LIN {X 0,Y 405.524,Z 705.596,A -85,B 0,C 180,E1 17049.688,E2 17049.688} C_VEL
LIN {X 0,Y 402.242,Z 726.337,A -85,B 0,C 180,E1 17048.422,E2 17048.422} C_VEL
LIN {X 0,Y 398.508,Z 746.053,A -85,B 0,C 180,E1 17046.936,E2 17046.936} C_VEL
LIN {X 0,Y 394.229,Z 765.506,A -85,B 0,C 180,E1 17045.152,E2 17045.152} C_VEL
LIN {X 0,Y 389.705,Z 783.802,A -85,B 0,C 180,E1 17043.128,E2 17043.128} C_VEL
LIN {X 0,Y 385.137,Z 800.764,A -85,B 0,C 180,E1 17040.878,E2 17040.878} C_VEL
LIN {X 0,Y 380.552,Z 816.747,A -85,B 0,C 180,E1 17038.332,E2 17038.332} C_VEL
LIN {X 0,Y 376.385,Z 830.752,A -85,B 0,C 180,E1 17035.659,E2 17035.659} C_VEL
LIN {X 0,Y 372.544,Z 843.468,A -85,B 0,C 180,E1 17032.736,E2 17032.736} C_VEL
LIN {X 0,Y 369.226,Z 854.588,A -85,B 0,C 180,E1 17029.621,E2 17029.621} C_VEL
LIN {X 0,Y 366.629,Z 863.669,A -85,B 0,C 180,E1 17026.477,E2 17026.477} C_VEL
LIN {X 0,Y 364.673,Z 871.061,A -85,B 0,C 180,E1 17023.251,E2 17023.251} C_VEL
LIN {X 0,Y 363.308,Z 876.769,A -85,B 0,C 180,E1 17019.985,E2 17019.985} C_VEL
LIN {X 0,Y 362.432,Z 881.033,A -85,B 0,C 180,E1 17016.495,E2 17016.495} C_VEL
LIN {X 0,Y 362.034,Z 883.325,A -85,B 0,C 180,E1 17013.417,E2 17013.417} C_VEL
LIN {X 0,Y 360.957,Z 883.954,A -85,B 0,C 180,E1 17012.201,E2 17012.201} C_VEL
LIN {X 0,Y 354.617,Z 885.109,A -85,B 0,C 180,E1 17008.857,E2 17008.857} C_VEL
LIN {X 0,Y 354.012,Z 884.908,A -85,B 0,C 180,E1 17007.87,E2 17007.87} C_VEL
LIN {X 0,Y 354.34,Z 883.134,A -85,B 0,C 180,E1 17004.495,E2 17004.495} C_VEL
LIN {X 0,Y 355.032,Z 879.694,A -85,B 0,C 180,E1 17001.089,E2 17001.089} C_VEL
LIN {X 0,Y 356.194,Z 874.854,A -85,B 0,C 180,E1 16997.846,E2 16997.846} C_VEL
LIN {X 0,Y 358.029,Z 868.036,A -85,B 0,C 180,E1 16994.449,E2 16994.449} C_VEL
LIN {X 0,Y 360.466,Z 859.76,A -85,B 0,C 180,E1 16991.23,E2 16991.23} C_VEL
LIN {X 0,Y 363.449,Z 850.138,A -85,B 0,C 180,E1 16988.198,E2 16988.198} C_VEL
LIN {X 0,Y 367.117,Z 838.547,A -85,B 0,C 180,E1 16985.201,E2 16985.201} C_VEL
LIN {X 0,Y 371.487,Z 824.659,A -85,B 0,C 180,E1 16982.248,E2 16982.248} C_VEL
LIN {X 0,Y 376.128,Z 809.477,A -85,B 0,C 180,E1 16979.574,E2 16979.574} C_VEL
LIN {X 0,Y 380.722,Z 793.669,A -85,B 0,C 180,E1 16977.247,E2 16977.247} C_VEL
LIN {X 0,Y 385.565,Z 775.624,A -85,B 0,C 180,E1 16975.032,E2 16975.032} C_VEL
LIN {X 0,Y 390.072,Z 757.084,A -85,B 0,C 180,E1 16973.143,E2 16973.143} C_VEL
LIN {X 0,Y 394.24,Z 737.467,A -85,B 0,C 180,E1 16971.49,E2 16971.49} C_VEL
LIN {X 0,Y 397.983,Z 716.674,A -85,B 0,C 180,E1 16970.065,E2 16970.065} C_VEL
LIN {X 0,Y 401.085,Z 695.03,A -85,B 0,C 180,E1 16968.883,E2 16968.883} C_VEL
LIN {X 0,Y 403.458,Z 672.77,A -85,B 0,C 180,E1 16967.951,E2 16967.951} C_VEL
LIN {X 0,Y 407.778,Z 629.715,A -85,B 0,C 180,E1 16966.545,E2 16966.545} C_VEL
LIN {X 0,Y 414.06,Z 571.27,A -85,B 0,C 180,E1 16964.995,E2 16964.995} C_VEL
LIN {X 0,Y 419.279,Z 512.395,A -85,B 0,C 180,E1 16963.682,E2 16963.682} C_VEL
LIN {X 0,Y 422.898,Z 458.138,A -85,B 0,C 180,E1 16962.666,E2 16962.666} C_VEL
LIN {X 0,Y 425.379,Z 415.515,A -85,B 0,C 180,E1 16961.93,E2 16961.93} C_VEL
LIN {X 0,Y 432.668,Z 383.274,A -85,B 0,C 180,E1 16960.762,E2 16960.762} C_VEL
LIN {X 0,Y 432.805,Z 378.392,A -85,B 0,C 180,E1 16960.393,E2 16960.393} C_VEL
LIN {X 0,Y 426.533,Z 360.369,A -85,B 0,C 180,E1 16957.723,E2 16957.723} C_VEL
LIN {X 0,Y 420.306,Z 344.672,A -85,B 0,C 180,E1 16955.079,E2 16955.079} C_VEL
LIN {X 0,Y 413.62,Z 329.35,A -85,B 0,C 180,E1 16952.129,E2 16952.129} C_VEL
LIN {X 0,Y 407.095,Z 316.323,A -85,B 0,C 180,E1 16949.26,E2 16949.26} C_VEL
LIN {X 0,Y 401.641,Z 306.431,A -85,B 0,C 180,E1 16946.783,E2 16946.783} C_VEL
LIN {X 0,Y 397.019,Z 298.327,A -85,B 0,C 180,E1 16944.475,E2 16944.475} C_VEL
LIN {X 0,Y 393.875,Z 293.356,A -85,B 0,C 180,E1 16942.934,E2 16942.934} C_VEL
LIN {X 0,Y 391.222,Z 288.934,A -85,B 0,C 180,E1 16941.437,E2 16941.437} C_VEL
LIN {X 0,Y 387.999,Z 284.027,A -85,B 0,C 180,E1 16939.652,E2 16939.652} C_VEL
LIN {X 0,Y 385.133,Z 279.626,A -85,B 0,C 180,E1 16937.879,E2 16937.879} C_VEL
LIN {X 0,Y 381.484,Z 274.487,A -85,B 0,C 180,E1 16935.429,E2 16935.429} C_VEL
LIN {X 0,Y 380.825,Z 273.211,A -85,B 0,C 180,E1 16934.91,E2 16934.91} C_VEL
LIN {X 0,Y 377.944,Z 270.024,A -85,B 0,C 180,E1 16932.762,E2 16932.762} C_VEL
LIN {X 0,Y 376.766,Z 267.259,A -85,B 0,C 180,E1 16931.481,E2 16931.481} C_VEL
LIN {X 0,Y 373.477,Z 264.326,A -85,B 0,C 180,E1 16928.468,E2 16928.468} C_VEL
LIN {X 0,Y 372.123,Z 260.992,A -85,B 0,C 180,E1 16926.325,E2 16926.325} C_VEL
LIN {X 0,Y 369.027,Z 258.675,A -85,B 0,C 180,E1 16918.758,E2 16918.758} C_VEL
LIN {X 0,Y 369.744,Z 259.37,A -85,B 0,C 180,E1 16914.102,E2 16914.102} C_VEL
LIN {X 0,Y 372.489,Z 261.356,A -85,B 0,C 180,E1 16909.561,E2 16909.561} C_VEL
LIN {X 0,Y 373.965,Z 268.68,A -85,B 0,C 180,E1 16906.824,E2 16906.824} C_VEL
LIN {X 0,Y 376.51,Z 277.821,A -85,B 0,C 180,E1 16903.809,E2 16903.809} C_VEL
LIN {X 0,Y 381.85,Z 292.334,A -85,B 0,C 180,E1 16899.619,E2 16899.619} C_VEL
LIN {X 0,Y 390.043,Z 308.671,A -85,B 0,C 180,E1 16895.946,E2 16895.946} C_VEL
LIN {X 0,Y 399.158,Z 327.437,A -85,B 0,C 180,E1 16892.161,E2 16892.161} C_VEL
LIN {X 0,Y 402.379,Z 333.924,A -85,B 0,C 180,E1 16890.99,E2 16890.99} C_VEL
LIN {X 0,Y 422.571,Z 365.09,A -85,B 0,C 180,E1 16887.399,E2 16887.399} C_VEL
LIN {X 0,Y 430.139,Z 377.336,A -85,B 0,C 180,E1 16886.138,E2 16886.138} C_VEL
LIN {X 0,Y 410.702,Z 628.411,A -85,B 0,C 180,E1 16880.76,E2 16880.76} C_VEL
LIN {X 0,Y 405.985,Z 693.922,A -85,B 0,C 180,E1 16879.282,E2 16879.282} C_VEL
LIN {X 0,Y 403.21,Z 718.115,A -85,B 0,C 180,E1 16878.518,E2 16878.518} C_VEL
LIN {X 0,Y 399.697,Z 742.919,A -85,B 0,C 180,E1 16877.489,E2 16877.489} C_VEL
LIN {X 0,Y 395.798,Z 766.429,A -85,B 0,C 180,E1 16876.262,E2 16876.262} C_VEL
LIN {X 0,Y 391.526,Z 788.691,A -85,B 0,C 180,E1 16874.818,E2 16874.818} C_VEL
LIN {X 0,Y 386.728,Z 811.509,A -85,B 0,C 180,E1 16873.045,E2 16873.045} C_VEL
LIN {X 0,Y 382.094,Z 831.899,A -85,B 0,C 180,E1 16871.158,E2 16871.158} C_VEL
LIN {X 0,Y 377.316,Z 851.634,A -85,B 0,C 180,E1 16868.998,E2 16868.998} C_VEL
LIN {X 0,Y 372.803,Z 869.858,A -85,B 0,C 180,E1 16866.683,E2 16866.683} C_VEL
LIN {X 0,Y 368.526,Z 886.743,A -85,B 0,C 180,E1 16864.154,E2 16864.154} C_VEL
LIN {X 0,Y 364.361,Z 903.466,A -85,B 0,C 180,E1 16861.242,E2 16861.242} C_VEL
LIN {X 0,Y 361.088,Z 917.18,A -85,B 0,C 180,E1 16858.443,E2 16858.443} C_VEL
LIN {X 0,Y 358.024,Z 931.1,A -85,B 0,C 180,E1 16855.119,E2 16855.119} C_VEL
LIN {X 0,Y 355.871,Z 942.358,A -85,B 0,C 180,E1 16851.943,E2 16851.943} C_VEL
LIN {X 0,Y 354.277,Z 952.735,A -85,B 0,C 180,E1 16848.427,E2 16848.427} C_VEL
LIN {X 0,Y 353.4,Z 960.861,A -85,B 0,C 180,E1 16845.088,E2 16845.088} C_VEL
LIN {X 0,Y 353.012,Z 967.793,A -85,B 0,C 180,E1 16841.469,E2 16841.469} C_VEL
LIN {X 0,Y 353.017,Z 972.197,A -85,B 0,C 180,E1 16838.47,E2 16838.47} C_VEL
LIN {X 0,Y 353.177,Z 975.815,A -85,B 0,C 180,E1 16835.035,E2 16835.035} C_VEL
LIN {X 0,Y 353.328,Z 977.637,A -85,B 0,C 180,E1 16831.784,E2 16831.784} C_VEL
LIN {X 0,Y 353.299,Z 978.106,A -85,B 0,C 180,E1 16828.865,E2 16828.865} C_VEL
LIN {X 0,Y 353.106,Z 977.399,A -85,B 0,C 180,E1 16825.778,E2 16825.778} C_VEL
LIN {X 0,Y 352.83,Z 975.02,A -85,B 0,C 180,E1 16822.182,E2 16822.182} C_VEL
LIN {X 0,Y 352.727,Z 971.431,A -85,B 0,C 180,E1 16818.886,E2 16818.886} C_VEL
LIN {X 0,Y 353.03,Z 966.335,A -85,B 0,C 180,E1 16815.399,E2 16815.399} C_VEL
LIN {X 0,Y 354.059,Z 959.013,A -85,B 0,C 180,E1 16811.561,E2 16811.561} C_VEL
LIN {X 0,Y 355.906,Z 950.42,A -85,B 0,C 180,E1 16807.885,E2 16807.885} C_VEL
LIN {X 0,Y 359.099,Z 939.101,A -85,B 0,C 180,E1 16803.9,E2 16803.9} C_VEL
LIN {X 0,Y 363.454,Z 926.402,A -85,B 0,C 180,E1 16800.136,E2 16800.136} C_VEL
LIN {X 0,Y 368.927,Z 912.1,A -85,B 0,C 180,E1 16796.592,E2 16796.592} C_VEL
LIN {X 0,Y 375.947,Z 895.333,A -85,B 0,C 180,E1 16793.052,E2 16793.052} C_VEL
LIN {X 0,Y 383.727,Z 877.917,A -85,B 0,C 180,E1 16789.938,E2 16789.938} C_VEL
LIN {X 0,Y 392.756,Z 858.185,A -85,B 0,C 180,E1 16786.977,E2 16786.977} C_VEL
LIN {X 0,Y 402.833,Z 836.606,A -85,B 0,C 180,E1 16784.266,E2 16784.266} C_VEL
LIN {X 0,Y 413.334,Z 814.204,A -85,B 0,C 180,E1 16781.938,E2 16781.938} C_VEL
LIN {X 0,Y 423.737,Z 791.887,A -85,B 0,C 180,E1 16780.029,E2 16780.029} C_VEL
LIN {X 0,Y 433.523,Z 770.179,A -85,B 0,C 180,E1 16778.516,E2 16778.516} C_VEL
LIN {X 0,Y 439.331,Z 756.867,A -85,B 0,C 180,E1 16777.71,E2 16777.71} C_VEL
LIN {X 0,Y 428.322,Z 776.559,A -85,B 0,C 180,E1 16776.284,E2 16776.284} C_VEL
LIN {X 0,Y 416.856,Z 796.27,A -85,B 0,C 180,E1 16774.478,E2 16774.478} C_VEL
LIN {X 0,Y 405.872,Z 815.235,A -85,B 0,C 180,E1 16772.316,E2 16772.316} C_VEL
LIN {X 0,Y 395.858,Z 832.952,A -85,B 0,C 180,E1 16769.841,E2 16769.841} C_VEL
LIN {X 0,Y 387.233,Z 848.533,A -85,B 0,C 180,E1 16767.196,E2 16767.196} C_VEL
LIN {X 0,Y 379.645,Z 862.38,A -85,B 0,C 180,E1 16764.317,E2 16764.317} C_VEL
LIN {X 0,Y 373.638,Z 873.294,A -85,B 0,C 180,E1 16761.508,E2 16761.508} C_VEL
LIN {X 0,Y 368.676,Z 882.065,A -85,B 0,C 180,E1 16758.665,E2 16758.665} C_VEL
LIN {X 0,Y 364.771,Z 888.63,A -85,B 0,C 180,E1 16755.909,E2 16755.909} C_VEL
LIN {X 0,Y 361.266,Z 893.892,A -85,B 0,C 180,E1 16752.792,E2 16752.792} C_VEL
LIN {X 0,Y 358.703,Z 896.947,A -85,B 0,C 180,E1 16749.79,E2 16749.79} C_VEL
LIN {X 0,Y 356.898,Z 898.104,A -85,B 0,C 180,E1 16746.919,E2 16746.919} C_VEL
LIN {X 0,Y 355.611,Z 897.569,A -85,B 0,C 180,E1 16744.031,E2 16744.031} C_VEL
LIN {X 0,Y 354.79,Z 895.361,A -85,B 0,C 180,E1 16741.13,E2 16741.13} C_VEL
LIN {X 0,Y 354.351,Z 891.466,A -85,B 0,C 180,E1 16738.221,E2 16738.221} C_VEL
LIN {X 0,Y 354.245,Z 885.77,A -85,B 0,C 180,E1 16735.305,E2 16735.305} C_VEL
LIN {X 0,Y 354.468,Z 878.694,A -85,B 0,C 180,E1 16732.544,E2 16732.544} C_VEL
LIN {X 0,Y 355.018,Z 869.756,A -85,B 0,C 180,E1 16729.779,E2 16729.779} C_VEL
LIN {X 0,Y 355.971,Z 858.79,A -85,B 0,C 180,E1 16727.014,E2 16727.014} C_VEL
LIN {X 0,Y 357.29,Z 846.403,A -85,B 0,C 180,E1 16724.415,E2 16724.415} C_VEL
LIN {X 0,Y 358.979,Z 832.235,A -85,B 0,C 180,E1 16721.919,E2 16721.919} C_VEL
LIN {X 0,Y 360.984,Z 816.384,A -85,B 0,C 180,E1 16719.573,E2 16719.573} C_VEL
LIN {X 0,Y 363.327,Z 798.388,A -85,B 0,C 180,E1 16717.338,E2 16717.338} C_VEL
LIN {X 0,Y 365.876,Z 778.547,A -85,B 0,C 180,E1 16715.283,E2 16715.283} C_VEL
LIN {X 0,Y 368.373,Z 758.536,A -85,B 0,C 180,E1 16713.567,E2 16713.567} C_VEL
LIN {X 0,Y 370.948,Z 736.616,A -85,B 0,C 180,E1 16712.029,E2 16712.029} C_VEL
LIN {X 0,Y 373.29,Z 714.104,A -85,B 0,C 180,E1 16710.779,E2 16710.779} C_VEL
LIN {X 0,Y 375.438,Z 690.485,A -85,B 0,C 180,E1 16709.778,E2 16709.778} C_VEL
LIN {X 0,Y 378.003,Z 654.561,A -85,B 0,C 180,E1 16708.688,E2 16708.688} C_VEL
LIN {X 0,Y 388.249,Z 512.214,A -85,B 0,C 180,E1 16704.784,E2 16704.784} C_VEL
LIN {X 0,Y 386.223,Z 472.757,A -85,B 0,C 180,E1 16703.224,E2 16703.224} C_VEL
LIN {X 0,Y 387.587,Z 472.354,A -85,B 0,C 180,E1 16702.959,E2 16702.959} C_VEL
LIN {X 0,Y 389.842,Z 469.038,A -85,B 0,C 180,E1 16702.61,E2 16702.61} C_VEL
LIN {X 0,Y 392.918,Z 461.347,A -85,B 0,C 180,E1 16702.241,E2 16702.241} C_VEL
LIN {X 0,Y 395.267,Z 453.532,A -85,B 0,C 180,E1 16702.023,E2 16702.023} C_VEL
LIN {X 0,Y 398.142,Z 449.735,A -85,B 0,C 180,E1 16701.591,E2 16701.591} C_VEL
LIN {X 0,Y 401.43,Z 442.671,A -85,B 0,C 180,E1 16701.189,E2 16701.189} C_VEL
LIN {X 0,Y 402.505,Z 440.316,A -85,B 0,C 180,E1 16701.061,E2 16701.061} C_VEL
LIN {X 0,Y 407.194,Z 436.824,A -85,B 0,C 180,E1 16700.324,E2 16700.324} C_VEL
LIN {X 0,Y 411.77,Z 431.891,A -85,B 0,C 180,E1 16699.674,E2 16699.674} C_VEL
LIN {X 0,Y 417.125,Z 427.794,A -85,B 0,C 180,E1 16698.897,E2 16698.897} C_VEL
LIN {X 0,Y 421.231,Z 423.838,A -85,B 0,C 180,E1 16698.345,E2 16698.345} C_VEL
LIN {X 0,Y 424.807,Z 421.477,A -85,B 0,C 180,E1 16697.849,E2 16697.849} C_VEL
LIN {X 0,Y 420.272,Z 497.691,A -85,B 0,C 180,E1 16696.51,E2 16696.51} C_VEL
LIN {X 0,Y 415.453,Z 555.616,A -85,B 0,C 180,E1 16695.271,E2 16695.271} C_VEL
LIN {X 0,Y 409.469,Z 613.57,A -85,B 0,C 180,E1 16693.806,E2 16693.806} C_VEL
LIN {X 0,Y 404.775,Z 657.664,A -85,B 0,C 180,E1 16692.472,E2 16692.472} C_VEL
LIN {X 0,Y 401.93,Z 687.022,A -85,B 0,C 180,E1 16691.373,E2 16691.373} C_VEL
LIN {X 0,Y 399.248,Z 707.767,A -85,B 0,C 180,E1 16690.346,E2 16690.346} C_VEL
LIN {X 0,Y 395.858,Z 728.321,A -85,B 0,C 180,E1 16689.066,E2 16689.066} C_VEL
LIN {X 0,Y 392.003,Z 747.896,A -85,B 0,C 180,E1 16687.562,E2 16687.562} C_VEL
LIN {X 0,Y 387.583,Z 767.232,A -85,B 0,C 180,E1 16685.756,E2 16685.756} C_VEL
LIN {X 0,Y 382.853,Z 785.607,A -85,B 0,C 180,E1 16683.682,E2 16683.682} C_VEL
LIN {X 0,Y 378.121,Z 802.479,A -85,B 0,C 180,E1 16681.396,E2 16681.396} C_VEL
LIN {X 0,Y 373.387,Z 818.314,A -85,B 0,C 180,E1 16678.818,E2 16678.818} C_VEL
LIN {X 0,Y 368.975,Z 832.505,A -85,B 0,C 180,E1 16676.041,E2 16676.041} C_VEL
LIN {X 0,Y 364.997,Z 845.109,A -85,B 0,C 180,E1 16673.063,E2 16673.063} C_VEL
LIN {X 0,Y 361.557,Z 856.127,A -85,B 0,C 180,E1 16669.887,E2 16669.887} C_VEL
LIN {X 0,Y 358.734,Z 865.576,A -85,B 0,C 180,E1 16666.499,E2 16666.499} C_VEL
LIN {X 0,Y 356.696,Z 872.928,A -85,B 0,C 180,E1 16663.124,E2 16663.124} C_VEL
LIN {X 0,Y 355.302,Z 878.489,A -85,B 0,C 180,E1 16659.721,E2 16659.721} C_VEL
LIN {X 0,Y 354.473,Z 882.337,A -85,B 0,C 180,E1 16656.316,E2 16656.316} C_VEL
LIN {X 0,Y 354.056,Z 884.554,A -85,B 0,C 180,E1 16652.914,E2 16652.914} C_VEL
LIN {X 0,Y 353.956,Z 885.197,A -85,B 0,C 180,E1 16649.676,E2 16649.676} C_VEL
LIN {X 0,Y 354.012,Z 884.908,A -85,B 0,C 180,E1 16647.87,E2 16647.87} C_VEL
LIN {X 0,Y 353.105,Z 884.552,A -85,B 0,C 180,E1 16646.622,E2 16646.622} C_VEL
LIN {X 0,Y 347.381,Z 883.219,A -85,B 0,C 180,E1 16643.272,E2 16643.272} C_VEL
LIN {X 0,Y 346.846,Z 882.204,A -85,B 0,C 180,E1 16642.185,E2 16642.185} C_VEL
LIN {X 0,Y 347.975,Z 877.54,A -85,B 0,C 180,E1 16638.564,E2 16638.564} C_VEL
LIN {X 0,Y 349.824,Z 870.903,A -85,B 0,C 180,E1 16634.924,E2 16634.924} C_VEL
LIN {X 0,Y 352.418,Z 862.388,A -85,B 0,C 180,E1 16631.377,E2 16631.377} C_VEL
LIN {X 0,Y 355.68,Z 852.278,A -85,B 0,C 180,E1 16628.044,E2 16628.044} C_VEL
LIN {X 0,Y 359.439,Z 840.872,A -85,B 0,C 180,E1 16624.986,E2 16624.986} C_VEL
LIN {X 0,Y 363.671,Z 828.008,A -85,B 0,C 180,E1 16622.134,E2 16622.134} C_VEL
LIN {X 0,Y 367.962,Z 814.594,A -85,B 0,C 180,E1 16619.64,E2 16619.64} C_VEL
LIN {X 0,Y 372.603,Z 799.462,A -85,B 0,C 180,E1 16617.267,E2 16617.267} C_VEL
LIN {X 0,Y 377.344,Z 782.911,A -85,B 0,C 180,E1 16615.085,E2 16615.085} C_VEL
LIN {X 0,Y 381.724,Z 766.258,A -85,B 0,C 180,E1 16613.235,E2 16613.235} C_VEL
LIN {X 0,Y 385.962,Z 748.26,A -85,B 0,C 180,E1 16611.556,E2 16611.556} C_VEL
LIN {X 0,Y 389.967,Z 728.551,A -85,B 0,C 180,E1 16610.037,E2 16610.037} C_VEL
LIN {X 0,Y 393.455,Z 707.895,A -85,B 0,C 180,E1 16608.75,E2 16608.75} C_VEL
LIN {X 0,Y 396.308,Z 686.094,A -85,B 0,C 180,E1 16607.682,E2 16607.682} C_VEL
LIN {X 0,Y 399.857,Z 650.548,A -85,B 0,C 180,E1 16606.387,E2 16606.387} C_VEL
LIN {X 0,Y 405.349,Z 601.675,A -85,B 0,C 180,E1 16604.956,E2 16604.956} C_VEL
LIN {X 0,Y 410.919,Z 547.326,A -85,B 0,C 180,E1 16603.616,E2 16603.616} C_VEL
LIN {X 0,Y 415.551,Z 490.609,A -85,B 0,C 180,E1 16602.431,E2 16602.431} C_VEL
LIN {X 0,Y 419.979,Z 418.206,A -85,B 0,C 180,E1 16601.155,E2 16601.155} C_VEL
LIN {X 0,Y 427.547,Z 384.988,A -85,B 0,C 180,E1 16599.96,E2 16599.96} C_VEL
LIN {X 0,Y 427.552,Z 382.519,A -85,B 0,C 180,E1 16599.764,E2 16599.764} C_VEL
LIN {X 0,Y 421.414,Z 364.665,A -85,B 0,C 180,E1 16597.061,E2 16597.061} C_VEL
LIN {X 0,Y 415.15,Z 348.657,A -85,B 0,C 180,E1 16594.298,E2 16594.298} C_VEL
LIN {X 0,Y 408.377,Z 333.351,A -85,B 0,C 180,E1 16591.27,E2 16591.27} C_VEL
LIN {X 0,Y 402.415,Z 321.186,A -85,B 0,C 180,E1 16588.494,E2 16588.494} C_VEL
LIN {X 0,Y 396.611,Z 310.397,A -85,B 0,C 180,E1 16585.698,E2 16585.698} C_VEL
LIN {X 0,Y 391.135,Z 301.045,A -85,B 0,C 180,E1 16582.866,E2 16582.866} C_VEL
LIN {X 0,Y 388.021,Z 295.874,A -85,B 0,C 180,E1 16581.068,E2 16581.068} C_VEL
LIN {X 0,Y 384.994,Z 291.173,A -85,B 0,C 180,E1 16579.338,E2 16579.338} C_VEL
LIN {X 0,Y 382.188,Z 286.545,A -85,B 0,C 180,E1 16577.47,E2 16577.47} C_VEL
LIN {X 0,Y 378.955,Z 282.176,A -85,B 0,C 180,E1 16575.299,E2 16575.299} C_VEL
LIN {X 0,Y 378.03,Z 280.526,A -85,B 0,C 180,E1 16574.553,E2 16574.553} C_VEL
LIN {X 0,Y 375.234,Z 277.05,A -85,B 0,C 180,E1 16572.309,E2 16572.309} C_VEL
LIN {X 0,Y 374.296,Z 274.809,A -85,B 0,C 180,E1 16571.245,E2 16571.245} C_VEL
LIN {X 0,Y 371.321,Z 271.937,A -85,B 0,C 180,E1 16568.283,E2 16568.283} C_VEL
LIN {X 0,Y 370.039,Z 268.706,A -85,B 0,C 180,E1 16566.205,E2 16566.205} C_VEL
LIN {X 0,Y 367.154,Z 266.442,A -85,B 0,C 180,E1 16558.596,E2 16558.596} C_VEL
LIN {X 0,Y 368.011,Z 267.237,A -85,B 0,C 180,E1 16553.917,E2 16553.917} C_VEL
LIN {X 0,Y 370.532,Z 269.088,A -85,B 0,C 180,E1 16549.819,E2 16549.819} C_VEL
LIN {X 0,Y 371.851,Z 275.876,A -85,B 0,C 180,E1 16547.262,E2 16547.262} C_VEL
LIN {X 0,Y 374.308,Z 285.032,A -85,B 0,C 180,E1 16544.228,E2 16544.228} C_VEL
LIN {X 0,Y 379.498,Z 300.184,A -85,B 0,C 180,E1 16539.849,E2 16539.849} C_VEL
LIN {X 0,Y 387.563,Z 319.875,A -85,B 0,C 180,E1 16535.132,E2 16535.132} C_VEL
LIN {X 0,Y 394.603,Z 335.094,A -85,B 0,C 180,E1 16532.004,E2 16532.004} C_VEL
LIN {X 0,Y 411.937,Z 361.642,A -85,B 0,C 180,E1 16528.807,E2 16528.807} C_VEL
LIN {X 0,Y 423.773,Z 380.727,A -85,B 0,C 180,E1 16526.766,E2 16526.766} C_VEL
LIN {X 0,Y 403.08,Z 640.594,A -85,B 0,C 180,E1 16521.094,E2 16521.094} C_VEL
LIN {X 0,Y 398.994,Z 694.506,A -85,B 0,C 180,E1 16519.834,E2 16519.834} C_VEL
LIN {X 0,Y 396.142,Z 718.636,A -85,B 0,C 180,E1 16519.054,E2 16519.054} C_VEL
LIN {X 0,Y 392.53,Z 743.375,A -85,B 0,C 180,E1 16518.002,E2 16518.002} C_VEL
LIN {X 0,Y 388.52,Z 766.895,A -85,B 0,C 180,E1 16516.746,E2 16516.746} C_VEL
LIN {X 0,Y 383.956,Z 790.092,A -85,B 0,C 180,E1 16515.205,E2 16515.205} C_VEL
LIN {X 0,Y 379.079,Z 812.597,A -85,B 0,C 180,E1 16513.402,E2 16513.402} C_VEL
LIN {X 0,Y 374.178,Z 833.62,A -85,B 0,C 180,E1 16511.405,E2 16511.405} C_VEL
LIN {X 0,Y 369.316,Z 853.128,A -85,B 0,C 180,E1 16509.19,E2 16509.19} C_VEL
LIN {X 0,Y 364.284,Z 872.858,A -85,B 0,C 180,E1 16506.557,E2 16506.557} C_VEL
LIN {X 0,Y 359.737,Z 890.512,A -85,B 0,C 180,E1 16503.79,E2 16503.79} C_VEL
LIN {X 0,Y 355.626,Z 906.727,A -85,B 0,C 180,E1 16500.778,E2 16500.778} C_VEL
LIN {X 0,Y 352.112,Z 921.437,A -85,B 0,C 180,E1 16497.572,E2 16497.572} C_VEL
LIN {X 0,Y 349.518,Z 933.352,A -85,B 0,C 180,E1 16494.507,E2 16494.507} C_VEL
LIN {X 0,Y 347.327,Z 945.157,A -85,B 0,C 180,E1 16490.914,E2 16490.914} C_VEL
LIN {X 0,Y 346.043,Z 954.062,A -85,B 0,C 180,E1 16487.662,E2 16487.662} C_VEL
LIN {X 0,Y 345.258,Z 962.402,A -85,B 0,C 180,E1 16483.908,E2 16483.908} C_VEL
LIN {X 0,Y 345.051,Z 967.893,A -85,B 0,C 180,E1 16480.778,E2 16480.778} C_VEL
LIN {X 0,Y 345.124,Z 972.521,A -85,B 0,C 180,E1 16477.324,E2 16477.324} C_VEL
LIN {X 0,Y 345.329,Z 975.386,A -85,B 0,C 180,E1 16473.985,E2 16473.985} C_VEL
LIN {X 0,Y 345.409,Z 976.769,A -85,B 0,C 180,E1 16470.995,E2 16470.995} C_VEL
LIN {X 0,Y 345.305,Z 977.005,A -85,B 0,C 180,E1 16467.843,E2 16467.843} C_VEL
LIN {X 0,Y 345.046,Z 975.752,A -85,B 0,C 180,E1 16464.346,E2 16464.346} C_VEL
LIN {X 0,Y 344.799,Z 973.147,A -85,B 0,C 180,E1 16460.991,E2 16460.991} C_VEL
LIN {X 0,Y 344.817,Z 969.073,A -85,B 0,C 180,E1 16457.439,E2 16457.439} C_VEL
LIN {X 0,Y 345.466,Z 962.594,A -85,B 0,C 180,E1 16453.349,E2 16453.349} C_VEL
LIN {X 0,Y 346.892,Z 955.072,A -85,B 0,C 180,E1 16449.588,E2 16449.588} C_VEL
LIN {X 0,Y 349.593,Z 944.98,A -85,B 0,C 180,E1 16445.498,E2 16445.498} C_VEL
LIN {X 0,Y 353.495,Z 933.505,A -85,B 0,C 180,E1 16441.606,E2 16441.606} C_VEL
LIN {X 0,Y 358.699,Z 920.105,A -85,B 0,C 180,E1 16437.831,E2 16437.831} C_VEL
LIN {X 0,Y 365.389,Z 904.751,A -85,B 0,C 180,E1 16434.153,E2 16434.153} C_VEL
LIN {X 0,Y 373.195,Z 888.055,A -85,B 0,C 180,E1 16430.779,E2 16430.779} C_VEL
LIN {X 0,Y 381.941,Z 870.073,A -85,B 0,C 180,E1 16427.716,E2 16427.716} C_VEL
LIN {X 0,Y 392.294,Z 849.528,A -85,B 0,C 180,E1 16424.777,E2 16424.777} C_VEL
LIN {X 0,Y 402.876,Z 828.807,A -85,B 0,C 180,E1 16422.302,E2 16422.302} C_VEL
LIN {X 0,Y 414.345,Z 806.273,A -85,B 0,C 180,E1 16420.095,E2 16420.095} C_VEL
LIN {X 0,Y 425.952,Z 783.125,A -85,B 0,C 180,E1 16418.259,E2 16418.259} C_VEL
LIN {X 0,Y 430.183,Z 774.498,A -85,B 0,C 180,E1 16417.663,E2 16417.663} C_VEL
LIN {X 0,Y 417.846,Z 793.984,A -85,B 0,C 180,E1 16415.978,E2 16415.978} C_VEL
LIN {X 0,Y 406.069,Z 812.314,A -85,B 0,C 180,E1 16413.984,E2 16413.984} C_VEL
LIN {X 0,Y 394.907,Z 829.925,A -85,B 0,C 180,E1 16411.609,E2 16411.609} C_VEL
LIN {X 0,Y 384.787,Z 846.339,A -85,B 0,C 180,E1 16408.903,E2 16408.903} C_VEL
LIN {X 0,Y 376.157,Z 860.63,A -85,B 0,C 180,E1 16406.015,E2 16406.015} C_VEL
LIN {X 0,Y 369.175,Z 872.195,A -85,B 0,C 180,E1 16403.124,E2 16403.124} C_VEL
LIN {X 0,Y 363.564,Z 881.294,A -85,B 0,C 180,E1 16400.275,E2 16400.275} C_VEL
LIN {X 0,Y 358.867,Z 888.538,A -85,B 0,C 180,E1 16397.345,E2 16397.345} C_VEL
LIN {X 0,Y 355.002,Z 893.969,A -85,B 0,C 180,E1 16394.326,E2 16394.326} C_VEL
LIN {X 0,Y 352.008,Z 897.518,A -85,B 0,C 180,E1 16391.303,E2 16391.303} C_VEL
LIN {X 0,Y 349.838,Z 899.205,A -85,B 0,C 180,E1 16388.382,E2 16388.382} C_VEL
LIN {X 0,Y 348.25,Z 899.262,A -85,B 0,C 180,E1 16385.437,E2 16385.437} C_VEL
LIN {X 0,Y 347.127,Z 897.443,A -85,B 0,C 180,E1 16382.311,E2 16382.311} C_VEL
LIN {X 0,Y 346.52,Z 893.961,A -85,B 0,C 180,E1 16379.339,E2 16379.339} C_VEL
LIN {X 0,Y 346.278,Z 889.094,A -85,B 0,C 180,E1 16376.524,E2 16376.524} C_VEL
LIN {X 0,Y 346.374,Z 882.169,A -85,B 0,C 180,E1 16373.536,E2 16373.536} C_VEL
LIN {X 0,Y 346.843,Z 873.252,A -85,B 0,C 180,E1 16370.542,E2 16370.542} C_VEL
LIN {X 0,Y 347.693,Z 862.814,A -85,B 0,C 180,E1 16367.713,E2 16367.713} C_VEL
LIN {X 0,Y 349.005,Z 850.164,A -85,B 0,C 180,E1 16364.888,E2 16364.888} C_VEL
LIN {X 0,Y 350.714,Z 835.834,A -85,B 0,C 180,E1 16362.221,E2 16362.221} C_VEL
LIN {X 0,Y 352.82,Z 819.581,A -85,B 0,C 180,E1 16359.686,E2 16359.686} C_VEL
LIN {X 0,Y 355.155,Z 802.162,A -85,B 0,C 180,E1 16357.408,E2 16357.408} C_VEL
LIN {X 0,Y 357.618,Z 783.595,A -85,B 0,C 180,E1 16355.38,E2 16355.38} C_VEL
LIN {X 0,Y 360.204,Z 763.387,A -85,B 0,C 180,E1 16353.542,E2 16353.542} C_VEL
LIN {X 0,Y 362.917,Z 741.169,A -85,B 0,C 180,E1 16351.892,E2 16351.892} C_VEL
LIN {X 0,Y 365.401,Z 718.55,A -85,B 0,C 180,E1 16350.547,E2 16350.547} C_VEL
LIN {X 0,Y 367.676,Z 694.971,A -85,B 0,C 180,E1 16349.467,E2 16349.467} C_VEL
LIN {X 0,Y 369.734,Z 668.465,A -85,B 0,C 180,E1 16348.594,E2 16348.594} C_VEL
LIN {X 0,Y 381.298,Z 513.044,A -85,B 0,C 180,E1 16344.201,E2 16344.201} C_VEL
LIN {X 0,Y 380.562,Z 497.793,A -85,B 0,C 180,E1 16343.573,E2 16343.573} C_VEL
LIN {X 0,Y 381.91,Z 497.424,A -85,B 0,C 180,E1 16343.302,E2 16343.302} C_VEL
LIN {X 0,Y 384.062,Z 494.38,A -85,B 0,C 180,E1 16342.96,E2 16342.96} C_VEL
LIN {X 0,Y 387.078,Z 487.132,A -85,B 0,C 180,E1 16342.589,E2 16342.589} C_VEL
LIN {X 0,Y 389.611,Z 478.921,A -85,B 0,C 180,E1 16342.352,E2 16342.352} C_VEL
LIN {X 0,Y 392.602,Z 474.92,A -85,B 0,C 180,E1 16341.893,E2 16341.893} C_VEL
LIN {X 0,Y 395.882,Z 467.794,A -85,B 0,C 180,E1 16341.483,E2 16341.483} C_VEL
LIN {X 0,Y 399.162,Z 458.109,A -85,B 0,C 180,E1 16341.157,E2 16341.157} C_VEL
LIN {X 0,Y 402.818,Z 452.307,A -85,B 0,C 180,E1 16340.661,E2 16340.661} C_VEL
LIN {X 0,Y 405.644,Z 446.453,A -85,B 0,C 180,E1 16340.326,E2 16340.326} C_VEL
LIN {X 0,Y 410.988,Z 441.796,A -85,B 0,C 180,E1 16339.535,E2 16339.535} C_VEL
LIN {X 0,Y 414.182,Z 438.511,A -85,B 0,C 180,E1 16339.093,E2 16339.093} C_VEL
LIN {X 0,Y 418.775,Z 435.159,A -85,B 0,C 180,E1 16338.439,E2 16338.439} C_VEL
LIN {X 0,Y 414.552,Z 502.765,A -85,B 0,C 180,E1 16337.229,E2 16337.229} C_VEL
LIN {X 0,Y 409.675,Z 559.247,A -85,B 0,C 180,E1 16336.005,E2 16336.005} C_VEL
LIN {X 0,Y 403.386,Z 618.02,A -85,B 0,C 180,E1 16334.497,E2 16334.497} C_VEL
LIN {X 0,Y 398.632,Z 661.485,A -85,B 0,C 180,E1 16333.138,E2 16333.138} C_VEL
LIN {X 0,Y 395.816,Z 689.205,A -85,B 0,C 180,E1 16332.072,E2 16332.072} C_VEL
LIN {X 0,Y 393.023,Z 709.908,A -85,B 0,C 180,E1 16331.024,E2 16331.024} C_VEL
LIN {X 0,Y 389.526,Z 730.303,A -85,B 0,C 180,E1 16329.73,E2 16329.73} C_VEL
LIN {X 0,Y 385.519,Z 749.859,A -85,B 0,C 180,E1 16328.199,E2 16328.199} C_VEL
LIN {X 0,Y 380.981,Z 768.959,A -85,B 0,C 180,E1 16326.38,E2 16326.38} C_VEL
LIN {X 0,Y 376.142,Z 787.06,A -85,B 0,C 180,E1 16324.302,E2 16324.302} C_VEL
LIN {X 0,Y 371.346,Z 803.534,A -85,B 0,C 180,E1 16322.036,E2 16322.036} C_VEL
LIN {X 0,Y 366.423,Z 819.368,A -85,B 0,C 180,E1 16319.418,E2 16319.418} C_VEL
LIN {X 0,Y 361.821,Z 833.553,A -85,B 0,C 180,E1 16316.595,E2 16316.595} C_VEL
LIN {X 0,Y 357.662,Z 846.148,A -85,B 0,C 180,E1 16313.564,E2 16313.564} C_VEL
LIN {X 0,Y 354.056,Z 857.156,A -85,B 0,C 180,E1 16310.326,E2 16310.326} C_VEL
LIN {X 0,Y 351.093,Z 866.569,A -85,B 0,C 180,E1 16306.881,E2 16306.881} C_VEL
LIN {X 0,Y 348.93,Z 873.941,A -85,B 0,C 180,E1 16303.422,E2 16303.422} C_VEL
LIN {X 0,Y 347.453,Z 879.498,A -85,B 0,C 180,E1 16299.943,E2 16299.943} C_VEL
LIN {X 0,Y 346.57,Z 883.344,A -85,B 0,C 180,E1 16296.461,E2 16296.461} C_VEL
LIN {X 0,Y 346.126,Z 885.557,A -85,B 0,C 180,E1 16292.981,E2 16292.981} C_VEL
LIN {X 0,Y 346.019,Z 886.198,A -85,B 0,C 180,E1 16289.669,E2 16289.669} C_VEL
LIN {X 0,Y 346.194,Z 885.284,A -85,B 0,C 180,E1 16286.191,E2 16286.191} C_VEL
LIN {X 0,Y 346.722,Z 882.699,A -85,B 0,C 180,E1 16282.71,E2 16282.71} C_VEL
LIN {X 0,Y 346.846,Z 882.204,A -85,B 0,C 180,E1 16282.185,E2 16282.185} C_VEL
LIN {X 0,Y 346.156,Z 880.919,A -85,B 0,C 180,E1 16280.926,E2 16280.926} C_VEL
LIN {X 0,Y 341.298,Z 877.302,A -85,B 0,C 180,E1 16277.623,E2 16277.623} C_VEL
LIN {X 0,Y 341.041,Z 875.505,A -85,B 0,C 180,E1 16276.445,E2 16276.445} C_VEL
LIN {X 0,Y 343.368,Z 867.961,A -85,B 0,C 180,E1 16272.774,E2 16272.774} C_VEL
LIN {X 0,Y 346.501,Z 858.52,A -85,B 0,C 180,E1 16269.21,E2 16269.21} C_VEL
LIN {X 0,Y 350.265,Z 847.584,A -85,B 0,C 180,E1 16265.907,E2 16265.907} C_VEL
LIN {X 0,Y 354.598,Z 835.063,A -85,B 0,C 180,E1 16262.819,E2 16262.819} C_VEL
LIN {X 0,Y 359.499,Z 820.631,A -85,B 0,C 180,E1 16259.883,E2 16259.883} C_VEL
LIN {X 0,Y 364.654,Z 804.731,A -85,B 0,C 180,E1 16257.211,E2 16257.211} C_VEL
LIN {X 0,Y 369.81,Z 787.687,A -85,B 0,C 180,E1 16254.837,E2 16254.837} C_VEL
LIN {X 0,Y 374.841,Z 769.486,A -85,B 0,C 180,E1 16252.734,E2 16252.734} C_VEL
LIN {X 0,Y 379.577,Z 750.118,A -85,B 0,C 180,E1 16250.884,E2 16250.884} C_VEL
LIN {X 0,Y 383.71,Z 730.552,A -85,B 0,C 180,E1 16249.348,E2 16249.348} C_VEL
LIN {X 0,Y 387.39,Z 709.552,A -85,B 0,C 180,E1 16248.018,E2 16248.018} C_VEL
LIN {X 0,Y 390.342,Z 687.798,A -85,B 0,C 180,E1 16246.936,E2 16246.936} C_VEL
LIN {X 0,Y 394.08,Z 651.812,A -85,B 0,C 180,E1 16245.605,E2 16245.605} C_VEL
LIN {X 0,Y 399.63,Z 604.047,A -85,B 0,C 180,E1 16244.183,E2 16244.183} C_VEL
LIN {X 0,Y 405.331,Z 550.107,A -85,B 0,C 180,E1 16242.839,E2 16242.839} C_VEL
LIN {X 0,Y 410.073,Z 493.875,A -85,B 0,C 180,E1 16241.652,E2 16241.652} C_VEL
LIN {X 0,Y 414.662,Z 421.018,A -85,B 0,C 180,E1 16240.361,E2 16240.361} C_VEL
LIN {X 0,Y 422.447,Z 386.912,A -85,B 0,C 180,E1 16239.152,E2 16239.152} C_VEL
LIN {X 0,Y 416.547,Z 369.52,A -85,B 0,C 180,E1 16236.473,E2 16236.473} C_VEL
LIN {X 0,Y 410.555,Z 353.951,A -85,B 0,C 180,E1 16233.731,E2 16233.731} C_VEL
LIN {X 0,Y 403.937,Z 338.684,A -85,B 0,C 180,E1 16230.659,E2 16230.659} C_VEL
LIN {X 0,Y 397.815,Z 326.026,A -85,B 0,C 180,E1 16227.71,E2 16227.71} C_VEL
LIN {X 0,Y 391.735,Z 314.733,A -85,B 0,C 180,E1 16224.626,E2 16224.626} C_VEL
LIN {X 0,Y 387.346,Z 307.149,A -85,B 0,C 180,E1 16222.221,E2 16222.221} C_VEL
LIN {X 0,Y 384.831,Z 302.805,A -85,B 0,C 180,E1 16220.693,E2 16220.693} C_VEL
LIN {X 0,Y 381.89,Z 298.168,A -85,B 0,C 180,E1 16218.945,E2 16218.945} C_VEL
LIN {X 0,Y 378.815,Z 293.128,A -85,B 0,C 180,E1 16216.8,E2 16216.8} C_VEL
LIN {X 0,Y 376.044,Z 288.933,A -85,B 0,C 180,E1 16214.789,E2 16214.789} C_VEL
LIN {X 0,Y 375.141,Z 287.663,A -85,B 0,C 180,E1 16214.037,E2 16214.037} C_VEL
LIN {X 0,Y 372.535,Z 283.918,A -85,B 0,C 180,E1 16211.77,E2 16211.77} C_VEL
LIN {X 0,Y 371.837,Z 282.354,A -85,B 0,C 180,E1 16211.007,E2 16211.007} C_VEL
LIN {X 0,Y 369.033,Z 279.335,A -85,B 0,C 180,E1 16207.943,E2 16207.943} C_VEL
LIN {X 0,Y 367.973,Z 276.423,A -85,B 0,C 180,E1 16206.083,E2 16206.083} C_VEL
LIN {X 0,Y 365.363,Z 274.251,A -85,B 0,C 180,E1 16198.745,E2 16198.745} C_VEL
LIN {X 0,Y 366.194,Z 274.958,A -85,B 0,C 180,E1 16194.202,E2 16194.202} C_VEL
LIN {X 0,Y 368.615,Z 276.787,A -85,B 0,C 180,E1 16190.081,E2 16190.081} C_VEL
LIN {X 0,Y 369.762,Z 283.067,A -85,B 0,C 180,E1 16187.705,E2 16187.705} C_VEL
LIN {X 0,Y 372.082,Z 292.23,A -85,B 0,C 180,E1 16184.651,E2 16184.651} C_VEL
LIN {X 0,Y 376.983,Z 307.006,A -85,B 0,C 180,E1 16180.355,E2 16180.355} C_VEL
LIN {X 0,Y 384.709,Z 326.553,A -85,B 0,C 180,E1 16175.631,E2 16175.631} C_VEL
LIN {X 0,Y 391.347,Z 341.571,A -85,B 0,C 180,E1 16172.516,E2 16172.516} C_VEL
LIN {X 0,Y 393.247,Z 345.859,A -85,B 0,C 180,E1 16171.796,E2 16171.796} C_VEL
LIN {X 0,Y 412.614,Z 375.965,A -85,B 0,C 180,E1 16168.251,E2 16168.251} C_VEL
LIN {X 0,Y 417.438,Z 384.037,A -85,B 0,C 180,E1 16167.41,E2 16167.41} C_VEL
LIN {X 0,Y 395.572,Z 650.308,A -85,B 0,C 180,E1 16161.48,E2 16161.48} C_VEL
LIN {X 0,Y 392.035,Z 694.97,A -85,B 0,C 180,E1 16160.405,E2 16160.405} C_VEL
LIN {X 0,Y 389.157,Z 718.638,A -85,B 0,C 180,E1 16159.623,E2 16159.623} C_VEL
LIN {X 0,Y 385.477,Z 743.215,A -85,B 0,C 180,E1 16158.559,E2 16158.559} C_VEL
LIN {X 0,Y 381.496,Z 766.089,A -85,B 0,C 180,E1 16157.323,E2 16157.323} C_VEL
LIN {X 0,Y 377.045,Z 788.248,A -85,B 0,C 180,E1 16155.835,E2 16155.835} C_VEL
LIN {X 0,Y 371.839,Z 811.835,A -85,B 0,C 180,E1 16153.929,E2 16153.929} C_VEL
LIN {X 0,Y 366.828,Z 832.877,A -85,B 0,C 180,E1 16151.899,E2 16151.899} C_VEL
LIN {X 0,Y 361.884,Z 852.27,A -85,B 0,C 180,E1 16149.662,E2 16149.662} C_VEL
LIN {X 0,Y 356.722,Z 872.11,A -85,B 0,C 180,E1 16146.979,E2 16146.979} C_VEL
LIN {X 0,Y 352.014,Z 889.979,A -85,B 0,C 180,E1 16144.125,E2 16144.125} C_VEL
LIN {X 0,Y 347.3,Z 908.742,A -85,B 0,C 180,E1 16140.636,E2 16140.636} C_VEL
LIN {X 0,Y 344.138,Z 921.897,A -85,B 0,C 180,E1 16137.702,E2 16137.702} C_VEL
LIN {X 0,Y 341.349,Z 934.307,A -85,B 0,C 180,E1 16134.357,E2 16134.357} C_VEL
LIN {X 0,Y 339.31,Z 944.889,A -85,B 0,C 180,E1 16130.889,E2 16130.889} C_VEL
LIN {X 0,Y 337.85,Z 955.285,A -85,B 0,C 180,E1 16126.86,E2 16126.86} C_VEL
LIN {X 0,Y 337.264,Z 962.477,A -85,B 0,C 180,E1 16123.37,E2 16123.37} C_VEL
LIN {X 0,Y 337.127,Z 968.432,A -85,B 0,C 180,E1 16119.733,E2 16119.733} C_VEL
LIN {X 0,Y 337.281,Z 972.371,A -85,B 0,C 180,E1 16116.297,E2 16116.297} C_VEL
LIN {X 0,Y 337.444,Z 974.7,A -85,B 0,C 180,E1 16113.227,E2 16113.227} C_VEL
LIN {X 0,Y 337.483,Z 975.907,A -85,B 0,C 180,E1 16110,E2 16110} C_VEL
LIN {X 0,Y 337.293,Z 975.724,A -85,B 0,C 180,E1 16106.601,E2 16106.601} C_VEL
LIN {X 0,Y 336.994,Z 974.236,A -85,B 0,C 180,E1 16103.355,E2 16103.355} C_VEL
LIN {X 0,Y 336.797,Z 971.576,A -85,B 0,C 180,E1 16100.085,E2 16100.085} C_VEL
LIN {X 0,Y 336.949,Z 966.726,A -85,B 0,C 180,E1 16096.018,E2 16096.018} C_VEL
LIN {X 0,Y 337.782,Z 960.62,A -85,B 0,C 180,E1 16092.248,E2 16092.248} C_VEL
LIN {X 0,Y 339.63,Z 952.598,A -85,B 0,C 180,E1 16088.226,E2 16088.226} C_VEL
LIN {X 0,Y 342.657,Z 942.693,A -85,B 0,C 180,E1 16084.228,E2 16084.228} C_VEL
LIN {X 0,Y 347.253,Z 930.62,A -85,B 0,C 180,E1 16080.123,E2 16080.123} C_VEL
LIN {X 0,Y 353.116,Z 917.09,A -85,B 0,C 180,E1 16076.289,E2 16076.289} C_VEL
LIN {X 0,Y 360.941,Z 900.734,A -85,B 0,C 180,E1 16072.4,E2 16072.4} C_VEL
LIN {X 0,Y 369.877,Z 883.356,A -85,B 0,C 180,E1 16068.936,E2 16068.936} C_VEL
LIN {X 0,Y 380.006,Z 864.49,A -85,B 0,C 180,E1 16065.791,E2 16065.791} C_VEL
LIN {X 0,Y 391.274,Z 843.862,A -85,B 0,C 180,E1 16062.933,E2 16062.933} C_VEL
LIN {X 0,Y 403.382,Z 822.083,A -85,B 0,C 180,E1 16060.449,E2 16060.449} C_VEL
LIN {X 0,Y 415.815,Z 799.709,A -85,B 0,C 180,E1 16058.379,E2 16058.379} C_VEL
LIN {X 0,Y 421.054,Z 790.222,A -85,B 0,C 180,E1 16057.612,E2 16057.612} C_VEL
LIN {X 0,Y 408.407,Z 808.115,A -85,B 0,C 180,E1 16055.813,E2 16055.813} C_VEL
LIN {X 0,Y 395.922,Z 825.807,A -85,B 0,C 180,E1 16053.579,E2 16053.579} C_VEL
LIN {X 0,Y 384.504,Z 842.367,A -85,B 0,C 180,E1 16050.99,E2 16050.99} C_VEL
LIN {X 0,Y 374.661,Z 856.99,A -85,B 0,C 180,E1 16048.189,E2 16048.189} C_VEL
LIN {X 0,Y 366.267,Z 869.642,A -85,B 0,C 180,E1 16045.206,E2 16045.206} C_VEL
LIN {X 0,Y 359.178,Z 880.187,A -85,B 0,C 180,E1 16042.075,E2 16042.075} C_VEL
LIN {X 0,Y 353.543,Z 888.234,A -85,B 0,C 180,E1 16038.98,E2 16038.98} C_VEL
LIN {X 0,Y 348.923,Z 894.302,A -85,B 0,C 180,E1 16035.797,E2 16035.797} C_VEL
LIN {X 0,Y 345.265,Z 898.383,A -85,B 0,C 180,E1 16032.545,E2 16032.545} C_VEL
LIN {X 0,Y 342.501,Z 900.474,A -85,B 0,C 180,E1 16029.24,E2 16029.24} C_VEL
LIN {X 0,Y 340.605,Z 900.563,A -85,B 0,C 180,E1 16026.067,E2 16026.067} C_VEL
LIN {X 0,Y 339.39,Z 898.942,A -85,B 0,C 180,E1 16023.04,E2 16023.04} C_VEL
LIN {X 0,Y 338.659,Z 895.626,A -85,B 0,C 180,E1 16020,E2 16020} C_VEL
LIN {X 0,Y 338.323,Z 890.618,A -85,B 0,C 180,E1 16016.951,E2 16016.951} C_VEL
LIN {X 0,Y 338.355,Z 884.258,A -85,B 0,C 180,E1 16014.063,E2 16014.063} C_VEL
LIN {X 0,Y 338.728,Z 876.113,A -85,B 0,C 180,E1 16011.17,E2 16011.17} C_VEL
LIN {X 0,Y 339.498,Z 866.06,A -85,B 0,C 180,E1 16008.275,E2 16008.275} C_VEL
LIN {X 0,Y 340.735,Z 853.868,A -85,B 0,C 180,E1 16005.382,E2 16005.382} C_VEL
LIN {X 0,Y 342.364,Z 840.096,A -85,B 0,C 180,E1 16002.669,E2 16002.669} C_VEL
LIN {X 0,Y 344.487,Z 823.708,A -85,B 0,C 180,E1 15999.971,E2 15999.971} C_VEL
LIN {X 0,Y 346.888,Z 806.117,A -85,B 0,C 180,E1 15997.547,E2 15997.547} C_VEL
LIN {X 0,Y 349.557,Z 786.744,A -85,B 0,C 180,E1 15995.315,E2 15995.315} C_VEL
LIN {X 0,Y 352.282,Z 766.215,A -85,B 0,C 180,E1 15993.355,E2 15993.355} C_VEL
LIN {X 0,Y 354.894,Z 745.696,A -85,B 0,C 180,E1 15991.749,E2 15991.749} C_VEL
LIN {X 0,Y 357.48,Z 723.115,A -85,B 0,C 180,E1 15990.325,E2 15990.325} C_VEL
LIN {X 0,Y 359.936,Z 699.006,A -85,B 0,C 180,E1 15989.144,E2 15989.144} C_VEL
LIN {X 0,Y 361.994,Z 674.681,A -85,B 0,C 180,E1 15988.269,E2 15988.269} C_VEL
LIN {X 0,Y 373.543,Z 526.866,A -85,B 0,C 180,E1 15983.969,E2 15983.969} C_VEL
LIN {X 0,Y 374.749,Z 526.346,A -85,B 0,C 180,E1 15983.725,E2 15983.725} C_VEL
LIN {X 0,Y 377.145,Z 522.135,A -85,B 0,C 180,E1 15983.379,E2 15983.379} C_VEL
LIN {X 0,Y 382.359,Z 508.589,A -85,B 0,C 180,E1 15982.802,E2 15982.802} C_VEL
LIN {X 0,Y 383.808,Z 503.98,A -85,B 0,C 180,E1 15982.673,E2 15982.673} C_VEL
LIN {X 0,Y 386.767,Z 500.125,A -85,B 0,C 180,E1 15982.214,E2 15982.214} C_VEL
LIN {X 0,Y 390.129,Z 493.051,A -85,B 0,C 180,E1 15981.795,E2 15981.795} C_VEL
LIN {X 0,Y 393.434,Z 483.485,A -85,B 0,C 180,E1 15981.466,E2 15981.466} C_VEL
LIN {X 0,Y 397.09,Z 477.73,A -85,B 0,C 180,E1 15980.962,E2 15980.962} C_VEL
LIN {X 0,Y 400.819,Z 469.022,A -85,B 0,C 180,E1 15980.542,E2 15980.542} C_VEL
LIN {X 0,Y 403.182,Z 462.32,A -85,B 0,C 180,E1 15980.312,E2 15980.312} C_VEL
LIN {X 0,Y 407.332,Z 455.185,A -85,B 0,C 180,E1 15979.789,E2 15979.789} C_VEL
LIN {X 0,Y 408.702,Z 452.461,A -85,B 0,C 180,E1 15979.63,E2 15979.63} C_VEL
LIN {X 0,Y 412.767,Z 449.062,A -85,B 0,C 180,E1 15979.043,E2 15979.043} C_VEL
LIN {X 0,Y 408.905,Z 507.719,A -85,B 0,C 180,E1 15977.97,E2 15977.97} C_VEL
LIN {X 0,Y 403.965,Z 562.831,A -85,B 0,C 180,E1 15976.759,E2 15976.759} C_VEL
LIN {X 0,Y 397.6,Z 620.328,A -85,B 0,C 180,E1 15975.263,E2 15975.263} C_VEL
LIN {X 0,Y 392.747,Z 663.489,A -85,B 0,C 180,E1 15973.889,E2 15973.889} C_VEL
LIN {X 0,Y 389.778,Z 691.389,A -85,B 0,C 180,E1 15972.794,E2 15972.794} C_VEL
LIN {X 0,Y 386.8,Z 712.442,A -85,B 0,C 180,E1 15971.703,E2 15971.703} C_VEL
LIN {X 0,Y 383.19,Z 732.554,A -85,B 0,C 180,E1 15970.396,E2 15970.396} C_VEL
LIN {X 0,Y 379.142,Z 751.575,A -85,B 0,C 180,E1 15968.878,E2 15968.878} C_VEL
LIN {X 0,Y 374.611,Z 769.999,A -85,B 0,C 180,E1 15967.101,E2 15967.101} C_VEL
LIN {X 0,Y 369.599,Z 788.112,A -85,B 0,C 180,E1 15964.997,E2 15964.997} C_VEL
LIN {X 0,Y 364.456,Z 805.095,A -85,B 0,C 180,E1 15962.62,E2 15962.62} C_VEL
LIN {X 0,Y 359.5,Z 820.419,A -85,B 0,C 180,E1 15960.043,E2 15960.043} C_VEL
LIN {X 0,Y 354.702,Z 834.6,A -85,B 0,C 180,E1 15957.173,E2 15957.173} C_VEL
LIN {X 0,Y 350.244,Z 847.507,A -85,B 0,C 180,E1 15953.999,E2 15953.999} C_VEL
LIN {X 0,Y 346.406,Z 858.676,A -85,B 0,C 180,E1 15950.619,E2 15950.619} C_VEL
LIN {X 0,Y 343.335,Z 867.971,A -85,B 0,C 180,E1 15947.106,E2 15947.106} C_VEL
LIN {X 0,Y 341.086,Z 875.281,A -85,B 0,C 180,E1 15943.563,E2 15943.563} C_VEL
LIN {X 0,Y 339.498,Z 880.979,A -85,B 0,C 180,E1 15939.836,E2 15939.836} C_VEL
LIN {X 0,Y 338.608,Z 884.646,A -85,B 0,C 180,E1 15936.273,E2 15936.273} C_VEL
LIN {X 0,Y 338.183,Z 886.622,A -85,B 0,C 180,E1 15932.881,E2 15932.881} C_VEL
LIN {X 0,Y 338.077,Z 887.155,A -85,B 0,C 180,E1 15929.322,E2 15929.322} C_VEL
LIN {X 0,Y 338.287,Z 886.201,A -85,B 0,C 180,E1 15925.932,E2 15925.932} C_VEL
LIN {X 0,Y 338.874,Z 883.559,A -85,B 0,C 180,E1 15922.37,E2 15922.37} C_VEL
LIN {X 0,Y 339.952,Z 879.257,A -85,B 0,C 180,E1 15918.807,E2 15918.807} C_VEL
LIN {X 0,Y 341.041,Z 875.505,A -85,B 0,C 180,E1 15916.445,E2 15916.445} C_VEL
LIN {X 0,Y 340.777,Z 873.444,A -85,B 0,C 180,E1 15915.189,E2 15915.189} C_VEL
LIN {X 0,Y 336.924,Z 867.433,A -85,B 0,C 180,E1 15911.803,E2 15911.803} C_VEL
LIN {X 0,Y 337.099,Z 865.021,A -85,B 0,C 180,E1 15910.743,E2 15910.743} C_VEL
LIN {X 0,Y 340.514,Z 855.39,A -85,B 0,C 180,E1 15907.377,E2 15907.377} C_VEL
LIN {X 0,Y 344.323,Z 844.841,A -85,B 0,C 180,E1 15904.362,E2 15904.362} C_VEL
LIN {X 0,Y 348.823,Z 832.357,A -85,B 0,C 180,E1 15901.4,E2 15901.4} C_VEL
LIN {X 0,Y 353.805,Z 818.12,A -85,B 0,C 180,E1 15898.593,E2 15898.593} C_VEL
LIN {X 0,Y 359.142,Z 802.082,A -85,B 0,C 180,E1 15895.971,E2 15895.971} C_VEL
LIN {X 0,Y 364.411,Z 784.985,A -85,B 0,C 180,E1 15893.653,E2 15893.653} C_VEL
LIN {X 0,Y 369.446,Z 766.967,A -85,B 0,C 180,E1 15891.623,E2 15891.623} C_VEL
LIN {X 0,Y 374.158,Z 747.889,A -85,B 0,C 180,E1 15889.845,E2 15889.845} C_VEL
LIN {X 0,Y 378.247,Z 728.625,A -85,B 0,C 180,E1 15888.369,E2 15888.369} C_VEL
LIN {X 0,Y 381.733,Z 708.857,A -85,B 0,C 180,E1 15887.136,E2 15887.136} C_VEL
LIN {X 0,Y 384.554,Z 688.472,A -85,B 0,C 180,E1 15886.124,E2 15886.124} C_VEL
LIN {X 0,Y 388.931,Z 648.613,A -85,B 0,C 180,E1 15884.644,E2 15884.644} C_VEL
LIN {X 0,Y 394.759,Z 599.861,A -85,B 0,C 180,E1 15883.21,E2 15883.21} C_VEL
LIN {X 0,Y 400.823,Z 542.636,A -85,B 0,C 180,E1 15881.805,E2 15881.805} C_VEL
LIN {X 0,Y 405.199,Z 490.011,A -85,B 0,C 180,E1 15880.716,E2 15880.716} C_VEL
LIN {X 0,Y 409.427,Z 423.831,A -85,B 0,C 180,E1 15879.546,E2 15879.546} C_VEL
LIN {X 0,Y 417.121,Z 390.364,A -85,B 0,C 180,E1 15878.379,E2 15878.379} C_VEL
LIN {X 0,Y 411.349,Z 373.311,A -85,B 0,C 180,E1 15875.689,E2 15875.689} C_VEL
LIN {X 0,Y 405.097,Z 356.95,A -85,B 0,C 180,E1 15872.721,E2 15872.721} C_VEL
LIN {X 0,Y 398.971,Z 342.808,A -85,B 0,C 180,E1 15869.751,E2 15869.751} C_VEL
LIN {X 0,Y 393.349,Z 331.094,A -85,B 0,C 180,E1 15866.903,E2 15866.903} C_VEL
LIN {X 0,Y 387.688,Z 320.219,A -85,B 0,C 180,E1 15863.886,E2 15863.886} C_VEL
LIN {X 0,Y 382.254,Z 310.598,A -85,B 0,C 180,E1 15860.679,E2 15860.679} C_VEL
LIN {X 0,Y 378.856,Z 305.168,A -85,B 0,C 180,E1 15858.544,E2 15858.544} C_VEL
LIN {X 0,Y 376.111,Z 300.461,A -85,B 0,C 180,E1 15856.527,E2 15856.527} C_VEL
LIN {X 0,Y 373.364,Z 296.078,A -85,B 0,C 180,E1 15854.422,E2 15854.422} C_VEL
LIN {X 0,Y 370.31,Z 291.589,A -85,B 0,C 180,E1 15851.605,E2 15851.605} C_VEL
LIN {X 0,Y 369.546,Z 289.935,A -85,B 0,C 180,E1 15850.76,E2 15850.76} C_VEL
LIN {X 0,Y 366.73,Z 286.813,A -85,B 0,C 180,E1 15847.678,E2 15847.678} C_VEL
LIN {X 0,Y 365.789,Z 284.091,A -85,B 0,C 180,E1 15845.805,E2 15845.805} C_VEL
LIN {X 0,Y 363.563,Z 282.033,A -85,B 0,C 180,E1 15838.582,E2 15838.582} C_VEL
LIN {X 0,Y 364.542,Z 282.885,A -85,B 0,C 180,E1 15833.859,E2 15833.859} C_VEL
LIN {X 0,Y 366.736,Z 284.467,A -85,B 0,C 180,E1 15830.347,E2 15830.347} C_VEL
LIN {X 0,Y 367.714,Z 290.381,A -85,B 0,C 180,E1 15828.113,E2 15828.113} C_VEL
LIN {X 0,Y 369.906,Z 299.664,A -85,B 0,C 180,E1 15825,E2 15825} C_VEL
LIN {X 0,Y 374.555,Z 313.976,A -85,B 0,C 180,E1 15820.831,E2 15820.831} C_VEL
LIN {X 0,Y 381.95,Z 333.396,A -85,B 0,C 180,E1 15816.102,E2 15816.102} C_VEL
LIN {X 0,Y 388.176,Z 347.845,A -85,B 0,C 180,E1 15813.082,E2 15813.082} C_VEL
LIN {X 0,Y 391.642,Z 356.438,A -85,B 0,C 180,E1 15811.628,E2 15811.628} C_VEL
LIN {X 0,Y 408.949,Z 383.589,A -85,B 0,C 180,E1 15808.45,E2 15808.45} C_VEL
LIN {X 0,Y 411.089,Z 387.345,A -85,B 0,C 180,E1 15808.064,E2 15808.064} C_VEL
LIN {X 0,Y 388.289,Z 656.277,A -85,B 0,C 180,E1 15801.95,E2 15801.95} C_VEL
LIN {X 0,Y 385.05,Z 695.396,A -85,B 0,C 180,E1 15800.98,E2 15800.98} C_VEL
LIN {X 0,Y 382.056,Z 719.294,A -85,B 0,C 180,E1 15800.171,E2 15800.171} C_VEL
LIN {X 0,Y 378.337,Z 743.436,A -85,B 0,C 180,E1 15799.1,E2 15799.1} C_VEL
LIN {X 0,Y 374.217,Z 766.461,A -85,B 0,C 180,E1 15797.826,E2 15797.826} C_VEL
LIN {X 0,Y 369.521,Z 789.281,A -85,B 0,C 180,E1 15796.259,E2 15796.259} C_VEL
LIN {X 0,Y 364.429,Z 811.762,A -85,B 0,C 180,E1 15794.399,E2 15794.399} C_VEL
LIN {X 0,Y 359.316,Z 832.761,A -85,B 0,C 180,E1 15792.332,E2 15792.332} C_VEL
LIN {X 0,Y 354.097,Z 852.805,A -85,B 0,C 180,E1 15789.972,E2 15789.972} C_VEL
LIN {X 0,Y 346.781,Z 881.406,A -85,B 0,C 180,E1 15786.03,E2 15786.03} C_VEL
LIN {X 0,Y 342.86,Z 896.81,A -85,B 0,C 180,E1 15783.448,E2 15783.448} C_VEL
LIN {X 0,Y 338.998,Z 911.599,A -85,B 0,C 180,E1 15780.486,E2 15780.486} C_VEL
LIN {X 0,Y 335.686,Z 924.838,A -85,B 0,C 180,E1 15777.304,E2 15777.304} C_VEL
LIN {X 0,Y 332.982,Z 936.48,A -85,B 0,C 180,E1 15773.915,E2 15773.915} C_VEL
LIN {X 0,Y 331.021,Z 946.585,A -85,B 0,C 180,E1 15770.327,E2 15770.327} C_VEL
LIN {X 0,Y 329.819,Z 955.151,A -85,B 0,C 180,E1 15766.557,E2 15766.557} C_VEL
LIN {X 0,Y 329.294,Z 962.307,A -85,B 0,C 180,E1 15762.913,E2 15762.913} C_VEL
LIN {X 0,Y 329.222,Z 968.117,A -85,B 0,C 180,E1 15759.087,E2 15759.087} C_VEL
LIN {X 0,Y 329.397,Z 971.698,A -85,B 0,C 180,E1 15755.749,E2 15755.749} C_VEL
LIN {X 0,Y 329.533,Z 973.873,A -85,B 0,C 180,E1 15752.609,E2 15752.609} C_VEL
LIN {X 0,Y 329.516,Z 974.904,A -85,B 0,C 180,E1 15749.131,E2 15749.131} C_VEL
LIN {X 0,Y 329.284,Z 974.461,A -85,B 0,C 180,E1 15745.821,E2 15745.821} C_VEL
LIN {X 0,Y 328.974,Z 972.922,A -85,B 0,C 180,E1 15742.666,E2 15742.666} C_VEL
LIN {X 0,Y 328.789,Z 970.053,A -85,B 0,C 180,E1 15739.201,E2 15739.201} C_VEL
LIN {X 0,Y 329.104,Z 965.009,A -85,B 0,C 180,E1 15735.034,E2 15735.034} C_VEL
LIN {X 0,Y 330.194,Z 958.667,A -85,B 0,C 180,E1 15731.094,E2 15731.094} C_VEL
LIN {X 0,Y 332.774,Z 949.221,A -85,B 0,C 180,E1 15726.445,E2 15726.445} C_VEL
LIN {X 0,Y 336.528,Z 938.905,A -85,B 0,C 180,E1 15722.303,E2 15722.303} C_VEL
LIN {X 0,Y 342.051,Z 926.084,A -85,B 0,C 180,E1 15718.055,E2 15718.055} C_VEL
LIN {X 0,Y 349.14,Z 911.666,A -85,B 0,C 180,E1 15714.049,E2 15714.049} C_VEL
LIN {X 0,Y 357.559,Z 895.887,A -85,B 0,C 180,E1 15710.388,E2 15710.388} C_VEL
LIN {X 0,Y 367.552,Z 878.113,A -85,B 0,C 180,E1 15706.935,E2 15706.935} C_VEL
LIN {X 0,Y 379.193,Z 858.346,A -85,B 0,C 180,E1 15703.738,E2 15703.738} C_VEL
LIN {X 0,Y 391.474,Z 838.016,A -85,B 0,C 180,E1 15701.028,E2 15701.028} C_VEL
LIN {X 0,Y 403.978,Z 817.307,A -85,B 0,C 180,E1 15698.77,E2 15698.77} C_VEL
LIN {X 0,Y 411.753,Z 804.434,A -85,B 0,C 180,E1 15697.555,E2 15697.555} C_VEL
LIN {X 0,Y 398.634,Z 821.4,A -85,B 0,C 180,E1 15695.586,E2 15695.586} C_VEL
LIN {X 0,Y 385.793,Z 838.082,A -85,B 0,C 180,E1 15693.152,E2 15693.152} C_VEL
LIN {X 0,Y 374.09,Z 853.588,A -85,B 0,C 180,E1 15690.343,E2 15690.343} C_VEL
LIN {X 0,Y 364.083,Z 867.125,A -85,B 0,C 180,E1 15687.299,E2 15687.299} C_VEL
LIN {X 0,Y 355.97,Z 878.109,A -85,B 0,C 180,E1 15684.211,E2 15684.211} C_VEL
LIN {X 0,Y 349.411,Z 886.787,A -85,B 0,C 180,E1 15681.109,E2 15681.109} C_VEL
LIN {X 0,Y 344.031,Z 893.466,A -85,B 0,C 180,E1 15677.944,E2 15677.944} C_VEL
LIN {X 0,Y 339.839,Z 898.112,A -85,B 0,C 180,E1 15674.831,E2 15674.831} C_VEL
LIN {X 0,Y 336.371,Z 901.078,A -85,B 0,C 180,E1 15671.488,E2 15671.488} C_VEL
LIN {X 0,Y 333.814,Z 902.079,A -85,B 0,C 180,E1 15668.093,E2 15668.093} C_VEL
LIN {X 0,Y 332.101,Z 901.142,A -85,B 0,C 180,E1 15664.836,E2 15664.836} C_VEL
LIN {X 0,Y 331.064,Z 898.555,A -85,B 0,C 180,E1 15661.731,E2 15661.731} C_VEL
LIN {X 0,Y 330.493,Z 894.274,A -85,B 0,C 180,E1 15658.613,E2 15658.613} C_VEL
LIN {X 0,Y 330.32,Z 888.236,A -85,B 0,C 180,E1 15655.486,E2 15655.486} C_VEL
LIN {X 0,Y 330.554,Z 880.375,A -85,B 0,C 180,E1 15652.351,E2 15652.351} C_VEL
LIN {X 0,Y 331.211,Z 870.397,A -85,B 0,C 180,E1 15649.212,E2 15649.212} C_VEL
LIN {X 0,Y 332.307,Z 858.864,A -85,B 0,C 180,E1 15646.249,E2 15646.249} C_VEL
LIN {X 0,Y 333.832,Z 845.677,A -85,B 0,C 180,E1 15643.428,E2 15643.428} C_VEL
LIN {X 0,Y 335.666,Z 831.482,A -85,B 0,C 180,E1 15640.872,E2 15640.872} C_VEL
LIN {X 0,Y 337.998,Z 814.487,A -85,B 0,C 180,E1 15638.298,E2 15638.298} C_VEL
LIN {X 0,Y 340.647,Z 795.749,A -85,B 0,C 180,E1 15635.92,E2 15635.92} C_VEL
LIN {X 0,Y 343.389,Z 775.87,A -85,B 0,C 180,E1 15633.823,E2 15633.823} C_VEL
LIN {X 0,Y 346.177,Z 755.006,A -85,B 0,C 180,E1 15632.007,E2 15632.007} C_VEL
LIN {X 0,Y 349.023,Z 732.045,A -85,B 0,C 180,E1 15630.384,E2 15630.384} C_VEL
LIN {X 0,Y 351.626,Z 708.502,A -85,B 0,C 180,E1 15629.07,E2 15629.07} C_VEL
LIN {X 0,Y 353.892,Z 684.83,A -85,B 0,C 180,E1 15628.076,E2 15628.076} C_VEL
LIN {X 0,Y 363.226,Z 566.065,A -85,B 0,C 180,E1 15624.49,E2 15624.49} C_VEL
LIN {X 0,Y 364.398,Z 565.695,A -85,B 0,C 180,E1 15624.235,E2 15624.235} C_VEL
LIN {X 0,Y 366.736,Z 562.036,A -85,B 0,C 180,E1 15623.883,E2 15623.883} C_VEL
LIN {X 0,Y 370.609,Z 552.646,A -85,B 0,C 180,E1 15623.47,E2 15623.47} C_VEL
LIN {X 0,Y 375.797,Z 536.079,A -85,B 0,C 180,E1 15623.089,E2 15623.089} C_VEL
LIN {X 0,Y 376.934,Z 532.398,A -85,B 0,C 180,E1 15622.999,E2 15622.999} C_VEL
LIN {X 0,Y 379.856,Z 527.791,A -85,B 0,C 180,E1 15622.574,E2 15622.574} C_VEL
LIN {X 0,Y 385.485,Z 514.31,A -85,B 0,C 180,E1 15621.96,E2 15621.96} C_VEL
LIN {X 0,Y 387.528,Z 508.554,A -85,B 0,C 180,E1 15621.762,E2 15621.762} C_VEL
LIN {X 0,Y 391.2,Z 502.869,A -85,B 0,C 180,E1 15621.252,E2 15621.252} C_VEL
LIN {X 0,Y 395.047,Z 494.148,A -85,B 0,C 180,E1 15620.827,E2 15620.827} C_VEL
LIN {X 0,Y 397.385,Z 487.686,A -85,B 0,C 180,E1 15620.602,E2 15620.602} C_VEL
LIN {X 0,Y 401.539,Z 480.63,A -85,B 0,C 180,E1 15620.071,E2 15620.071} C_VEL
LIN {X 0,Y 405.657,Z 470.714,A -85,B 0,C 180,E1 15619.647,E2 15619.647} C_VEL
LIN {X 0,Y 406.476,Z 468.475,A -85,B 0,C 180,E1 15619.569,E2 15619.569} C_VEL
LIN {X 0,Y 402.319,Z 524.845,A -85,B 0,C 180,E1 15618.478,E2 15618.478} C_VEL
LIN {X 0,Y 396.817,Z 580.477,A -85,B 0,C 180,E1 15617.187,E2 15617.187} C_VEL
LIN {X 0,Y 390.225,Z 636.395,A -85,B 0,C 180,E1 15615.641,E2 15615.641} C_VEL
LIN {X 0,Y 385.459,Z 679.331,A -85,B 0,C 180,E1 15614.147,E2 15614.147} C_VEL
LIN {X 0,Y 382.827,Z 700.965,A -85,B 0,C 180,E1 15613.181,E2 15613.181} C_VEL
LIN {X 0,Y 379.315,Z 722.606,A -85,B 0,C 180,E1 15611.931,E2 15611.931} C_VEL
LIN {X 0,Y 375.208,Z 742.953,A -85,B 0,C 180,E1 15610.459,E2 15610.459} C_VEL
LIN {X 0,Y 370.621,Z 762.224,A -85,B 0,C 180,E1 15608.749,E2 15608.749} C_VEL
LIN {X 0,Y 365.496,Z 781.044,A -85,B 0,C 180,E1 15606.72,E2 15606.72} C_VEL
LIN {X 0,Y 360.132,Z 798.788,A -85,B 0,C 180,E1 15604.403,E2 15604.403} C_VEL
LIN {X 0,Y 355.054,Z 814.339,A -85,B 0,C 180,E1 15601.968,E2 15601.968} C_VEL
LIN {X 0,Y 349.757,Z 829.623,A -85,B 0,C 180,E1 15599.078,E2 15599.078} C_VEL
LIN {X 0,Y 345.024,Z 842.835,A -85,B 0,C 180,E1 15596.052,E2 15596.052} C_VEL
LIN {X 0,Y 340.799,Z 854.532,A -85,B 0,C 180,E1 15592.786,E2 15592.786} C_VEL
LIN {X 0,Y 337.298,Z 864.397,A -85,B 0,C 180,E1 15589.391,E2 15589.391} C_VEL
LIN {X 0,Y 334.407,Z 872.934,A -85,B 0,C 180,E1 15585.677,E2 15585.677} C_VEL
LIN {X 0,Y 332.397,Z 879.384,A -85,B 0,C 180,E1 15581.98,E2 15581.98} C_VEL
LIN {X 0,Y 331.13,Z 883.931,A -85,B 0,C 180,E1 15578.334,E2 15578.334} C_VEL
LIN {X 0,Y 330.454,Z 886.711,A -85,B 0,C 180,E1 15574.86,E2 15574.86} C_VEL
LIN {X 0,Y 330.158,Z 888.078,A -85,B 0,C 180,E1 15571.215,E2 15571.215} C_VEL
LIN {X 0,Y 330.21,Z 887.92,A -85,B 0,C 180,E1 15567.744,E2 15567.744} C_VEL
LIN {X 0,Y 330.607,Z 886.15,A -85,B 0,C 180,E1 15564.098,E2 15564.098} C_VEL
LIN {X 0,Y 331.45,Z 882.726,A -85,B 0,C 180,E1 15560.449,E2 15560.449} C_VEL
LIN {X 0,Y 332.921,Z 877.621,A -85,B 0,C 180,E1 15556.806,E2 15556.806} C_VEL
LIN {X 0,Y 335.132,Z 870.725,A -85,B 0,C 180,E1 15553.178,E2 15553.178} C_VEL
LIN {X 0,Y 337.099,Z 865.021,A -85,B 0,C 180,E1 15550.743,E2 15550.743} C_VEL
LIN {X 0,Y 337.28,Z 862.137,A -85,B 0,C 180,E1 15549.519,E2 15549.519} C_VEL
LIN {X 0,Y 334.683,Z 854.109,A -85,B 0,C 180,E1 15546.195,E2 15546.195} C_VEL
LIN {X 0,Y 335.215,Z 850.992,A -85,B 0,C 180,E1 15545.188,E2 15545.188} C_VEL
LIN {X 0,Y 339.668,Z 839.224,A -85,B 0,C 180,E1 15542.092,E2 15542.092} C_VEL
LIN {X 0,Y 344.597,Z 825.915,A -85,B 0,C 180,E1 15539.192,E2 15539.192} C_VEL
LIN {X 0,Y 349.831,Z 811.181,A -85,B 0,C 180,E1 15536.521,E2 15536.521} C_VEL
LIN {X 0,Y 355.241,Z 794.915,A -85,B 0,C 180,E1 15534.066,E2 15534.066} C_VEL
LIN {X 0,Y 360.526,Z 777.635,A -85,B 0,C 180,E1 15531.896,E2 15531.896} C_VEL
LIN {X 0,Y 365.555,Z 759.306,A -85,B 0,C 180,E1 15529.985,E2 15529.985} C_VEL
LIN {X 0,Y 370.087,Z 740.299,A -85,B 0,C 180,E1 15528.346,E2 15528.346} C_VEL
LIN {X 0,Y 373.931,Z 721.419,A -85,B 0,C 180,E1 15527.01,E2 15527.01} C_VEL
LIN {X 0,Y 377.231,Z 701.418,A -85,B 0,C 180,E1 15525.863,E2 15525.863} C_VEL
LIN {X 0,Y 379.945,Z 679.696,A -85,B 0,C 180,E1 15524.892,E2 15524.892} C_VEL
LIN {X 0,Y 384.883,Z 636.923,A -85,B 0,C 180,E1 15523.391,E2 15523.391} C_VEL
LIN {X 0,Y 391.604,Z 581.818,A -85,B 0,C 180,E1 15521.854,E2 15521.854} C_VEL
LIN {X 0,Y 397.135,Z 527.059,A -85,B 0,C 180,E1 15520.58,E2 15520.58} C_VEL
LIN {X 0,Y 401.186,Z 474.554,A -85,B 0,C 180,E1 15519.55,E2 15519.55} C_VEL
LIN {X 0,Y 404.446,Z 425.834,A -85,B 0,C 180,E1 15518.684,E2 15518.684} C_VEL
LIN {X 0,Y 411.795,Z 393.606,A -85,B 0,C 180,E1 15517.551,E2 15517.551} C_VEL
LIN {X 0,Y 406.174,Z 376.822,A -85,B 0,C 180,E1 15514.829,E2 15514.829} C_VEL
LIN {X 0,Y 400.038,Z 360.802,A -85,B 0,C 180,E1 15511.83,E2 15511.83} C_VEL
LIN {X 0,Y 394.105,Z 346.94,A -85,B 0,C 180,E1 15508.82,E2 15508.82} C_VEL
LIN {X 0,Y 388.507,Z 335.003,A -85,B 0,C 180,E1 15505.782,E2 15505.782} C_VEL
LIN {X 0,Y 383.362,Z 325.292,A -85,B 0,C 180,E1 15502.91,E2 15502.91} C_VEL
LIN {X 0,Y 378.832,Z 317.185,A -85,B 0,C 180,E1 15500.148,E2 15500.148} C_VEL
LIN {X 0,Y 376.064,Z 312.469,A -85,B 0,C 180,E1 15498.285,E2 15498.285} C_VEL
LIN {X 0,Y 373.303,Z 307.665,A -85,B 0,C 180,E1 15496.175,E2 15496.175} C_VEL
LIN {X 0,Y 370.356,Z 302.809,A -85,B 0,C 180,E1 15493.744,E2 15493.744} C_VEL
LIN {X 0,Y 367.881,Z 298.791,A -85,B 0,C 180,E1 15491.206,E2 15491.206} C_VEL
LIN {X 0,Y 367.263,Z 297.512,A -85,B 0,C 180,E1 15490.51,E2 15490.51} C_VEL
LIN {X 0,Y 364.554,Z 294.322,A -85,B 0,C 180,E1 15487.407,E2 15487.407} C_VEL
LIN {X 0,Y 363.716,Z 291.804,A -85,B 0,C 180,E1 15485.68,E2 15485.68} C_VEL
LIN {X 0,Y 361.663,Z 289.804,A -85,B 0,C 180,E1 15478.574,E2 15478.574} C_VEL
LIN {X 0,Y 362.753,Z 290.696,A -85,B 0,C 180,E1 15473.829,E2 15473.829} C_VEL
LIN {X 0,Y 364.756,Z 292.106,A -85,B 0,C 180,E1 15470.613,E2 15470.613} C_VEL
LIN {X 0,Y 365.624,Z 297.788,A -85,B 0,C 180,E1 15468.484,E2 15468.484} C_VEL
LIN {X 0,Y 367.843,Z 307.216,A -85,B 0,C 180,E1 15465.317,E2 15465.317} C_VEL
LIN {X 0,Y 372.203,Z 321.229,A -85,B 0,C 180,E1 15461.234,E2 15461.234} C_VEL
LIN {X 0,Y 379.349,Z 340.558,A -85,B 0,C 180,E1 15456.505,E2 15456.505} C_VEL
LIN {X 0,Y 385.038,Z 354.114,A -85,B 0,C 180,E1 15453.657,E2 15453.657} C_VEL
LIN {X 0,Y 390.121,Z 367.099,A -85,B 0,C 180,E1 15451.445,E2 15451.445} C_VEL
LIN {X 0,Y 404.754,Z 390.58,A -85,B 0,C 180,E1 15448.732,E2 15448.732} C_VEL
LIN {X 0,Y 382.202,Z 647.493,A -85,B 0,C 180,E1 15442.792,E2 15442.792} C_VEL
LIN {X 0,Y 378.254,Z 694.409,A -85,B 0,C 180,E1 15441.615,E2 15441.615} C_VEL
LIN {X 0,Y 375.199,Z 718.281,A -85,B 0,C 180,E1 15440.796,E2 15440.796} C_VEL
LIN {X 0,Y 371.43,Z 742.34,A -85,B 0,C 180,E1 15439.721,E2 15439.721} C_VEL
LIN {X 0,Y 367.2,Z 765.576,A -85,B 0,C 180,E1 15438.424,E2 15438.424} C_VEL
LIN {X 0,Y 362.344,Z 788.699,A -85,B 0,C 180,E1 15436.815,E2 15436.815} C_VEL
LIN {X 0,Y 357.035,Z 811.648,A -85,B 0,C 180,E1 15434.884,E2 15434.884} C_VEL
LIN {X 0,Y 351.826,Z 832.542,A -85,B 0,C 180,E1 15432.784,E2 15432.784} C_VEL
LIN {X 0,Y 344.9,Z 860.914,A -85,B 0,C 180,E1 15429.542,E2 15429.542} C_VEL
LIN {X 0,Y 340.515,Z 878.143,A -85,B 0,C 180,E1 15427.165,E2 15427.165} C_VEL
LIN {X 0,Y 336.3,Z 893.898,A -85,B 0,C 180,E1 15424.555,E2 15424.555} C_VEL
LIN {X 0,Y 332.196,Z 908.772,A -85,B 0,C 180,E1 15421.583,E2 15421.583} C_VEL
LIN {X 0,Y 328.571,Z 922.264,A -85,B 0,C 180,E1 15418.342,E2 15418.342} C_VEL
LIN {X 0,Y 325.611,Z 934.225,A -85,B 0,C 180,E1 15414.879,E2 15414.879} C_VEL
LIN {X 0,Y 323.409,Z 944.532,A -85,B 0,C 180,E1 15411.206,E2 15411.206} C_VEL
LIN {X 0,Y 322.001,Z 953.295,A -85,B 0,C 180,E1 15407.344,E2 15407.344} C_VEL
LIN {X 0,Y 321.334,Z 961.857,A -85,B 0,C 180,E1 15402.581,E2 15402.581} C_VEL
LIN {X 0,Y 321.31,Z 967.333,A -85,B 0,C 180,E1 15398.771,E2 15398.771} C_VEL
LIN {X 0,Y 321.501,Z 970.682,A -85,B 0,C 180,E1 15395.532,E2 15395.532} C_VEL
LIN {X 0,Y 321.63,Z 972.821,A -85,B 0,C 180,E1 15392.316,E2 15392.316} C_VEL
LIN {X 0,Y 321.586,Z 973.802,A -85,B 0,C 180,E1 15388.753,E2 15388.753} C_VEL
LIN {X 0,Y 321.29,Z 973.303,A -85,B 0,C 180,E1 15385.359,E2 15385.359} C_VEL
LIN {X 0,Y 320.963,Z 971.595,A -85,B 0,C 180,E1 15381.941,E2 15381.941} C_VEL
LIN {X 0,Y 320.822,Z 968.386,A -85,B 0,C 180,E1 15378.129,E2 15378.129} C_VEL
LIN {X 0,Y 321.357,Z 962.923,A -85,B 0,C 180,E1 15373.738,E2 15373.738} C_VEL
LIN {X 0,Y 322.761,Z 956.408,A -85,B 0,C 180,E1 15369.698,E2 15369.698} C_VEL
LIN {X 0,Y 325.715,Z 947.137,A -85,B 0,C 180,E1 15365.129,E2 15365.129} C_VEL
LIN {X 0,Y 330.29,Z 936.141,A -85,B 0,C 180,E1 15360.677,E2 15360.677} C_VEL
LIN {X 0,Y 336.456,Z 923.364,A -85,B 0,C 180,E1 15356.443,E2 15356.443} C_VEL
LIN {X 0,Y 345.049,Z 907.611,A -85,B 0,C 180,E1 15352.096,E2 15352.096} C_VEL
LIN {X 0,Y 354.861,Z 891.066,A -85,B 0,C 180,E1 15348.305,E2 15348.305} C_VEL
LIN {X 0,Y 366.402,Z 872.536,A -85,B 0,C 180,E1 15344.803,E2 15344.803} C_VEL
LIN {X 0,Y 379.135,Z 852.734,A -85,B 0,C 180,E1 15341.724,E2 15341.724} C_VEL
LIN {X 0,Y 393.5,Z 830.922,A -85,B 0,C 180,E1 15338.963,E2 15338.963} C_VEL
LIN {X 0,Y 402.533,Z 817.272,A -85,B 0,C 180,E1 15337.511,E2 15337.511} C_VEL
LIN {X 0,Y 388.816,Z 833.433,A -85,B 0,C 180,E1 15335.353,E2 15335.353} C_VEL
LIN {X 0,Y 375.59,Z 849.152,A -85,B 0,C 180,E1 15332.713,E2 15332.713} C_VEL
LIN {X 0,Y 364.132,Z 863.085,A -85,B 0,C 180,E1 15329.803,E2 15329.803} C_VEL
LIN {X 0,Y 354.32,Z 875.14,A -85,B 0,C 180,E1 15326.66,E2 15326.66} C_VEL
LIN {X 0,Y 346.379,Z 884.782,A -85,B 0,C 180,E1 15323.476,E2 15323.476} C_VEL
LIN {X 0,Y 339.731,Z 892.49,A -85,B 0,C 180,E1 15320.142,E2 15320.142} C_VEL
LIN {X 0,Y 334.529,Z 897.963,A -85,B 0,C 180,E1 15316.854,E2 15316.854} C_VEL
LIN {X 0,Y 330.569,Z 901.446,A -85,B 0,C 180,E1 15313.647,E2 15313.647} C_VEL
LIN {X 0,Y 327.503,Z 903.2,A -85,B 0,C 180,E1 15310.377,E2 15310.377} C_VEL
LIN {X 0,Y 325.153,Z 903.121,A -85,B 0,C 180,E1 15306.888,E2 15306.888} C_VEL
LIN {X 0,Y 323.645,Z 901.16,A -85,B 0,C 180,E1 15303.543,E2 15303.543} C_VEL
LIN {X 0,Y 322.794,Z 897.601,A -85,B 0,C 180,E1 15300.355,E2 15300.355} C_VEL
LIN {X 0,Y 322.388,Z 892.347,A -85,B 0,C 180,E1 15297.156,E2 15297.156} C_VEL
LIN {X 0,Y 322.4,Z 885.246,A -85,B 0,C 180,E1 15293.947,E2 15293.947} C_VEL
LIN {X 0,Y 322.842,Z 876.242,A -85,B 0,C 180,E1 15290.732,E2 15290.732} C_VEL
LIN {X 0,Y 323.708,Z 865.731,A -85,B 0,C 180,E1 15287.694,E2 15287.694} C_VEL
LIN {X 0,Y 325.083,Z 853,A -85,B 0,C 180,E1 15284.662,E2 15284.662} C_VEL
LIN {X 0,Y 326.885,Z 838.717,A -85,B 0,C 180,E1 15281.82,E2 15281.82} C_VEL
LIN {X 0,Y 329.147,Z 822.349,A -85,B 0,C 180,E1 15279.087,E2 15279.087} C_VEL
LIN {X 0,Y 331.661,Z 804.898,A -85,B 0,C 180,E1 15276.644,E2 15276.644} C_VEL
LIN {X 0,Y 334.416,Z 785.713,A -85,B 0,C 180,E1 15274.402,E2 15274.402} C_VEL
LIN {X 0,Y 337.334,Z 764.634,A -85,B 0,C 180,E1 15272.362,E2 15272.362} C_VEL
LIN {X 0,Y 340.268,Z 742.481,A -85,B 0,C 180,E1 15270.611,E2 15270.611} C_VEL
LIN {X 0,Y 343.05,Z 719.236,A -85,B 0,C 180,E1 15269.137,E2 15269.137} C_VEL
LIN {X 0,Y 345.561,Z 695.392,A -85,B 0,C 180,E1 15267.97,E2 15267.97} C_VEL
LIN {X 0,Y 347.887,Z 668.16,A -85,B 0,C 180,E1 15267.005,E2 15267.005} C_VEL
LIN {X 0,Y 353.235,Z 601.06,A -85,B 0,C 180,E1 15264.926,E2 15264.926} C_VEL
LIN {X 0,Y 354.377,Z 600.785,A -85,B 0,C 180,E1 15264.661,E2 15264.661} C_VEL
LIN {X 0,Y 356.658,Z 597.525,A -85,B 0,C 180,E1 15264.304,E2 15264.304} C_VEL
LIN {X 0,Y 360.359,Z 589.269,A -85,B 0,C 180,E1 15263.906,E2 15263.906} C_VEL
LIN {X 0,Y 365.374,Z 574.567,A -85,B 0,C 180,E1 15263.555,E2 15263.555} C_VEL
LIN {X 0,Y 366.315,Z 571.825,A -85,B 0,C 180,E1 15263.484,E2 15263.484} C_VEL
LIN {X 0,Y 369.232,Z 567.614,A -85,B 0,C 180,E1 15263.045,E2 15263.045} C_VEL
LIN {X 0,Y 373.102,Z 559.212,A -85,B 0,C 180,E1 15262.614,E2 15262.614} C_VEL
LIN {X 0,Y 378.287,Z 544.108,A -85,B 0,C 180,E1 15262.21,E2 15262.21} C_VEL
LIN {X 0,Y 380.664,Z 536.478,A -85,B 0,C 180,E1 15262.05,E2 15262.05} C_VEL
LIN {X 0,Y 384.336,Z 529.971,A -85,B 0,C 180,E1 15261.579,E2 15261.579} C_VEL
LIN {X 0,Y 390.486,Z 514.755,A -85,B 0,C 180,E1 15260.968,E2 15260.968} C_VEL
LIN {X 0,Y 391.377,Z 512.758,A -85,B 0,C 180,E1 15260.873,E2 15260.873} C_VEL
LIN {X 0,Y 395.569,Z 505.766,A -85,B 0,C 180,E1 15260.338,E2 15260.338} C_VEL
LIN {X 0,Y 399.483,Z 496.795,A -85,B 0,C 180,E1 15259.931,E2 15259.931} C_VEL
LIN {X 0,Y 394.883,Z 549.537,A -85,B 0,C 180,E1 15258.818,E2 15258.818} C_VEL
LIN {X 0,Y 388.84,Z 604.249,A -85,B 0,C 180,E1 15257.446,E2 15257.446} C_VEL
LIN {X 0,Y 383.007,Z 651.573,A -85,B 0,C 180,E1 15256.024,E2 15256.024} C_VEL
LIN {X 0,Y 378.619,Z 690.17,A -85,B 0,C 180,E1 15254.56,E2 15254.56} C_VEL
LIN {X 0,Y 375.677,Z 710.691,A -85,B 0,C 180,E1 15253.526,E2 15253.526} C_VEL
LIN {X 0,Y 371.933,Z 731.108,A -85,B 0,C 180,E1 15252.229,E2 15252.229} C_VEL
LIN {X 0,Y 367.522,Z 751.012,A -85,B 0,C 180,E1 15250.662,E2 15250.662} C_VEL
LIN {X 0,Y 362.643,Z 769.877,A -85,B 0,C 180,E1 15248.849,E2 15248.849} C_VEL
LIN {X 0,Y 357.426,Z 787.746,A -85,B 0,C 180,E1 15246.774,E2 15246.774} C_VEL
LIN {X 0,Y 352.005,Z 804.576,A -85,B 0,C 180,E1 15244.421,E2 15244.421} C_VEL
LIN {X 0,Y 346.71,Z 819.846,A -85,B 0,C 180,E1 15241.854,E2 15241.854} C_VEL
LIN {X 0,Y 341.668,Z 833.676,A -85,B 0,C 180,E1 15239.065,E2 15239.065} C_VEL
LIN {X 0,Y 336.758,Z 846.745,A -85,B 0,C 180,E1 15235.879,E2 15235.879} C_VEL
LIN {X 0,Y 332.441,Z 858.175,A -85,B 0,C 180,E1 15232.457,E2 15232.457} C_VEL
LIN {X 0,Y 328.822,Z 867.957,A -85,B 0,C 180,E1 15228.804,E2 15228.804} C_VEL
LIN {X 0,Y 326.036,Z 875.95,A -85,B 0,C 180,E1 15224.973,E2 15224.973} C_VEL
LIN {X 0,Y 324.137,Z 881.846,A -85,B 0,C 180,E1 15221.197,E2 15221.197} C_VEL
LIN {X 0,Y 322.991,Z 885.922,A -85,B 0,C 180,E1 15217.471,E2 15217.471} C_VEL
LIN {X 0,Y 322.411,Z 888.316,A -85,B 0,C 180,E1 15213.912,E2 15213.912} C_VEL
LIN {X 0,Y 322.213,Z 889.207,A -85,B 0,C 180,E1 15210.178,E2 15210.178} C_VEL
LIN {X 0,Y 322.344,Z 888.541,A -85,B 0,C 180,E1 15206.621,E2 15206.621} C_VEL
LIN {X 0,Y 322.894,Z 886.307,A -85,B 0,C 180,E1 15202.885,E2 15202.885} C_VEL
LIN {X 0,Y 323.974,Z 882.449,A -85,B 0,C 180,E1 15199.148,E2 15199.148} C_VEL
LIN {X 0,Y 325.657,Z 877.203,A -85,B 0,C 180,E1 15195.599,E2 15195.599} C_VEL
LIN {X 0,Y 328.184,Z 869.891,A -85,B 0,C 180,E1 15191.895,E2 15191.895} C_VEL
LIN {X 0,Y 331.613,Z 860.58,A -85,B 0,C 180,E1 15188.231,E2 15188.231} C_VEL
LIN {X 0,Y 335.215,Z 850.992,A -85,B 0,C 180,E1 15185.188,E2 15185.188} C_VEL
LIN {X 0,Y 335.806,Z 847.302,A -85,B 0,C 180,E1 15184.025,E2 15184.025} C_VEL
LIN {X 0,Y 334.369,Z 837.952,A -85,B 0,C 180,E1 15180.994,E2 15180.994} C_VEL
LIN {X 0,Y 335.24,Z 833.575,A -85,B 0,C 180,E1 15179.896,E2 15179.896} C_VEL
LIN {X 0,Y 340.501,Z 819.67,A -85,B 0,C 180,E1 15177.094,E2 15177.094} C_VEL
LIN {X 0,Y 345.707,Z 805.162,A -85,B 0,C 180,E1 15174.65,E2 15174.65} C_VEL
LIN {X 0,Y 351.333,Z 788.291,A -85,B 0,C 180,E1 15172.274,E2 15172.274} C_VEL
LIN {X 0,Y 356.785,Z 770.221,A -85,B 0,C 180,E1 15170.165,E2 15170.165} C_VEL
LIN {X 0,Y 361.814,Z 751.331,A -85,B 0,C 180,E1 15168.346,E2 15168.346} C_VEL
LIN {X 0,Y 366.386,Z 731.238,A -85,B 0,C 180,E1 15166.765,E2 15166.765} C_VEL
LIN {X 0,Y 370.253,Z 710.53,A -85,B 0,C 180,E1 15165.455,E2 15165.455} C_VEL
LIN {X 0,Y 373.355,Z 688.971,A -85,B 0,C 180,E1 15164.386,E2 15164.386} C_VEL
LIN {X 0,Y 378.118,Z 648.948,A -85,B 0,C 180,E1 15162.876,E2 15162.876} C_VEL
LIN {X 0,Y 384.174,Z 601.052,A -85,B 0,C 180,E1 15161.453,E2 15161.453} C_VEL
LIN {X 0,Y 390.361,Z 545.706,A -85,B 0,C 180,E1 15160.079,E2 15160.079} C_VEL
LIN {X 0,Y 394.842,Z 494.374,A -85,B 0,C 180,E1 15159.009,E2 15159.009} C_VEL
LIN {X 0,Y 399.349,Z 428.73,A -85,B 0,C 180,E1 15157.831,E2 15157.831} C_VEL
LIN {X 0,Y 406.606,Z 397.088,A -85,B 0,C 180,E1 15156.74,E2 15156.74} C_VEL
LIN {X 0,Y 401.35,Z 381.205,A -85,B 0,C 180,E1 15154.094,E2 15154.094} C_VEL
LIN {X 0,Y 395.659,Z 366.11,A -85,B 0,C 180,E1 15151.203,E2 15151.203} C_VEL
LIN {X 0,Y 390.132,Z 352.976,A -85,B 0,C 180,E1 15148.304,E2 15148.304} C_VEL
LIN {X 0,Y 384.975,Z 341.645,A -85,B 0,C 180,E1 15145.376,E2 15145.376} C_VEL
LIN {X 0,Y 380.102,Z 332.089,A -85,B 0,C 180,E1 15142.504,E2 15142.504} C_VEL
LIN {X 0,Y 375.733,Z 324.127,A -85,B 0,C 180,E1 15139.753,E2 15139.753} C_VEL
LIN {X 0,Y 373.065,Z 319.456,A -85,B 0,C 180,E1 15137.872,E2 15137.872} C_VEL
LIN {X 0,Y 370.614,Z 314.988,A -85,B 0,C 180,E1 15135.893,E2 15135.893} C_VEL
LIN {X 0,Y 367.877,Z 310.29,A -85,B 0,C 180,E1 15133.518,E2 15133.518} C_VEL
LIN {X 0,Y 365.476,Z 306.133,A -85,B 0,C 180,E1 15130.881,E2 15130.881} C_VEL
LIN {X 0,Y 364.988,Z 305.086,A -85,B 0,C 180,E1 15130.257,E2 15130.257} C_VEL
LIN {X 0,Y 362.386,Z 301.831,A -85,B 0,C 180,E1 15127.132,E2 15127.132} C_VEL
LIN {X 0,Y 361.666,Z 299.521,A -85,B 0,C 180,E1 15125.553,E2 15125.553} C_VEL
LIN {X 0,Y 359.843,Z 297.595,A -85,B 0,C 180,E1 15118.567,E2 15118.567} C_VEL
LIN {X 0,Y 361.042,Z 298.525,A -85,B 0,C 180,E1 15113.799,E2 15113.799} C_VEL
LIN {X 0,Y 362.837,Z 299.912,A -85,B 0,C 180,E1 15110.803,E2 15110.803} C_VEL
LIN {X 0,Y 364.105,Z 307.723,A -85,B 0,C 180,E1 15107.953,E2 15107.953} C_VEL
LIN {X 0,Y 366.044,Z 315.833,A -85,B 0,C 180,E1 15105.324,E2 15105.324} C_VEL
LIN {X 0,Y 369.783,Z 328.376,A -85,B 0,C 180,E1 15101.663,E2 15101.663} C_VEL
LIN {X 0,Y 376.578,Z 347.233,A -85,B 0,C 180,E1 15097.026,E2 15097.026} C_VEL
LIN {X 0,Y 381.903,Z 360.372,A -85,B 0,C 180,E1 15094.239,E2 15094.239} C_VEL
LIN {X 0,Y 388.582,Z 377.895,A -85,B 0,C 180,E1 15091.258,E2 15091.258} C_VEL
LIN {X 0,Y 398.412,Z 393.907,A -85,B 0,C 180,E1 15089.409,E2 15089.409} C_VEL
LIN {X 0,Y 373.667,Z 668.611,A -85,B 0,C 180,E1 15082.908,E2 15082.908} C_VEL
LIN {X 0,Y 370.77,Z 698.909,A -85,B 0,C 180,E1 15082.082,E2 15082.082} C_VEL
LIN {X 0,Y 367.548,Z 722.861,A -85,B 0,C 180,E1 15081.212,E2 15081.212} C_VEL
LIN {X 0,Y 363.541,Z 746.89,A -85,B 0,C 180,E1 15080.057,E2 15080.057} C_VEL
LIN {X 0,Y 358.932,Z 770.714,A -85,B 0,C 180,E1 15078.625,E2 15078.625} C_VEL
LIN {X 0,Y 354.087,Z 792.961,A -85,B 0,C 180,E1 15077.002,E2 15077.002} C_VEL
LIN {X 0,Y 348.844,Z 814.672,A -85,B 0,C 180,E1 15075.07,E2 15075.07} C_VEL
LIN {X 0,Y 342.947,Z 841.315,A -85,B 0,C 180,E1 15072.564,E2 15072.564} C_VEL
LIN {X 0,Y 338.565,Z 859.044,A -85,B 0,C 180,E1 15070.521,E2 15070.521} C_VEL
LIN {X 0,Y 334.073,Z 875.956,A -85,B 0,C 180,E1 15068.175,E2 15068.175} C_VEL
LIN {X 0,Y 329.719,Z 891.424,A -85,B 0,C 180,E1 15065.609,E2 15065.609} C_VEL
LIN {X 0,Y 325.413,Z 906.23,A -85,B 0,C 180,E1 15062.657,E2 15062.657} C_VEL
LIN {X 0,Y 321.568,Z 919.684,A -85,B 0,C 180,E1 15059.425,E2 15059.425} C_VEL
LIN {X 0,Y 318.306,Z 931.885,A -85,B 0,C 180,E1 15055.89,E2 15055.89} C_VEL
LIN {X 0,Y 315.936,Z 942.016,A -85,B 0,C 180,E1 15052.32,E2 15052.32} C_VEL
LIN {X 0,Y 314.285,Z 951.055,A -85,B 0,C 180,E1 15048.359,E2 15048.359} C_VEL
LIN {X 0,Y 313.503,Z 958.173,A -85,B 0,C 180,E1 15044.405,E2 15044.405} C_VEL
LIN {X 0,Y 313.371,Z 965.46,A -85,B 0,C 180,E1 15039.365,E2 15039.365} C_VEL
LIN {X 0,Y 313.578,Z 969.332,A -85,B 0,C 180,E1 15035.673,E2 15035.673} C_VEL
LIN {X 0,Y 313.718,Z 971.463,A -85,B 0,C 180,E1 15032.557,E2 15032.557} C_VEL
LIN {X 0,Y 313.699,Z 972.514,A -85,B 0,C 180,E1 15029.452,E2 15029.452} C_VEL
LIN {X 0,Y 313.427,Z 972.468,A -85,B 0,C 180,E1 15025.975,E2 15025.975} C_VEL
LIN {X 0,Y 313.02,Z 970.857,A -85,B 0,C 180,E1 15022.105,E2 15022.105} C_VEL
LIN {X 0,Y 312.839,Z 967.991,A -85,B 0,C 180,E1 15018.383,E2 15018.383} C_VEL
LIN {X 0,Y 313.249,Z 963.47,A -85,B 0,C 180,E1 15014.257,E2 15014.257} C_VEL
LIN {X 0,Y 314.719,Z 956.729,A -85,B 0,C 180,E1 15009.738,E2 15009.738} C_VEL
LIN {X 0,Y 317.559,Z 948.375,A -85,B 0,C 180,E1 15005.243,E2 15005.243} C_VEL
LIN {X 0,Y 322.2,Z 937.7,A -85,B 0,C 180,E1 15000.638,E2 15000.638} C_VEL
LIN {X 0,Y 328.995,Z 924.676,A -85,B 0,C 180,E1 14995.998,E2 14995.998} C_VEL
LIN {X 0,Y 337.596,Z 910.093,A -85,B 0,C 180,E1 14991.71,E2 14991.71} C_VEL
LIN {X 0,Y 347.982,Z 893.721,A -85,B 0,C 180,E1 14987.749,E2 14987.749} C_VEL
LIN {X 0,Y 360.429,Z 875.269,A -85,B 0,C 180,E1 14984.068,E2 14984.068} C_VEL
LIN {X 0,Y 373.911,Z 856.085,A -85,B 0,C 180,E1 14980.932,E2 14980.932} C_VEL
LIN {X 0,Y 389.053,Z 835.026,A -85,B 0,C 180,E1 14978.146,E2 14978.146} C_VEL
LIN {X 0,Y 393.229,Z 829.126,A -85,B 0,C 180,E1 14977.457,E2 14977.457} C_VEL
LIN {X 0,Y 378.6,Z 844.84,A -85,B 0,C 180,E1 14975.043,E2 14975.043} C_VEL
LIN {X 0,Y 364.829,Z 859.877,A -85,B 0,C 180,E1 14972.12,E2 14972.12} C_VEL
LIN {X 0,Y 353.199,Z 872.771,A -85,B 0,C 180,E1 14968.953,E2 14968.953} C_VEL
LIN {X 0,Y 343.722,Z 883.267,A -85,B 0,C 180,E1 14965.686,E2 14965.686} C_VEL
LIN {X 0,Y 336.086,Z 891.463,A -85,B 0,C 180,E1 14962.384,E2 14962.384} C_VEL
LIN {X 0,Y 330.01,Z 897.493,A -85,B 0,C 180,E1 14959.101,E2 14959.101} C_VEL
LIN {X 0,Y 325.055,Z 901.743,A -85,B 0,C 180,E1 14955.706,E2 14955.706} C_VEL
LIN {X 0,Y 321.344,Z 904.085,A -85,B 0,C 180,E1 14952.398,E2 14952.398} C_VEL
LIN {X 0,Y 318.546,Z 904.725,A -85,B 0,C 180,E1 14949.03,E2 14949.03} C_VEL
LIN {X 0,Y 316.543,Z 903.592,A -85,B 0,C 180,E1 14945.62,E2 14945.62} C_VEL
LIN {X 0,Y 315.25,Z 900.615,A -85,B 0,C 180,E1 14942.181,E2 14942.181} C_VEL
LIN {X 0,Y 314.585,Z 896.074,A -85,B 0,C 180,E1 14938.907,E2 14938.907} C_VEL
LIN {X 0,Y 314.363,Z 889.809,A -85,B 0,C 180,E1 14935.622,E2 14935.622} C_VEL
LIN {X 0,Y 314.561,Z 882.135,A -85,B 0,C 180,E1 14932.511,E2 14932.511} C_VEL
LIN {X 0,Y 315.17,Z 872.642,A -85,B 0,C 180,E1 14929.397,E2 14929.397} C_VEL
LIN {X 0,Y 316.272,Z 861.168,A -85,B 0,C 180,E1 14926.284,E2 14926.284} C_VEL
LIN {X 0,Y 317.81,Z 848.196,A -85,B 0,C 180,E1 14923.363,E2 14923.363} C_VEL
LIN {X 0,Y 319.873,Z 832.797,A -85,B 0,C 180,E1 14920.46,E2 14920.46} C_VEL
LIN {X 0,Y 322.331,Z 815.748,A -85,B 0,C 180,E1 14917.762,E2 14917.762} C_VEL
LIN {X 0,Y 325.123,Z 796.996,A -85,B 0,C 180,E1 14915.275,E2 14915.275} C_VEL
LIN {X 0,Y 328.019,Z 777.192,A -85,B 0,C 180,E1 14913.085,E2 14913.085} C_VEL
LIN {X 0,Y 330.97,Z 756.171,A -85,B 0,C 180,E1 14911.178,E2 14911.178} C_VEL
LIN {X 0,Y 333.937,Z 733.443,A -85,B 0,C 180,E1 14909.501,E2 14909.501} C_VEL
LIN {X 0,Y 336.653,Z 710.193,A -85,B 0,C 180,E1 14908.139,E2 14908.139} C_VEL
LIN {X 0,Y 339.159,Z 685.708,A -85,B 0,C 180,E1 14907.048,E2 14907.048} C_VEL
LIN {X 0,Y 343.478,Z 632.653,A -85,B 0,C 180,E1 14905.311,E2 14905.311} C_VEL
LIN {X 0,Y 344.735,Z 632.45,A -85,B 0,C 180,E1 14905,E2 14905} C_VEL
LIN {X 0,Y 347.033,Z 629.365,A -85,B 0,C 180,E1 14904.633,E2 14904.633} C_VEL
LIN {X 0,Y 350.778,Z 621.496,A -85,B 0,C 180,E1 14904.23,E2 14904.23} C_VEL
LIN {X 0,Y 355.643,Z 608.037,A -85,B 0,C 180,E1 14903.913,E2 14903.913} C_VEL
LIN {X 0,Y 356.115,Z 606.902,A -85,B 0,C 180,E1 14903.869,E2 14903.869} C_VEL
LIN {X 0,Y 359.151,Z 602.741,A -85,B 0,C 180,E1 14903.406,E2 14903.406} C_VEL
LIN {X 0,Y 363.027,Z 594.841,A -85,B 0,C 180,E1 14902.983,E2 14902.983} C_VEL
LIN {X 0,Y 368.138,Z 580.915,A -85,B 0,C 180,E1 14902.605,E2 14902.605} C_VEL
LIN {X 0,Y 369.769,Z 576.111,A -85,B 0,C 180,E1 14902.5,E2 14902.5} C_VEL
LIN {X 0,Y 373.573,Z 569.906,A -85,B 0,C 180,E1 14902.004,E2 14902.004} C_VEL
LIN {X 0,Y 378.079,Z 559.492,A -85,B 0,C 180,E1 14901.562,E2 14901.562} C_VEL
LIN {X 0,Y 383.632,Z 542.779,A -85,B 0,C 180,E1 14901.188,E2 14901.188} C_VEL
LIN {X 0,Y 384.603,Z 540.122,A -85,B 0,C 180,E1 14901.108,E2 14901.108} C_VEL
LIN {X 0,Y 388.796,Z 532.262,A -85,B 0,C 180,E1 14900.623,E2 14900.623} C_VEL
LIN {X 0,Y 392.244,Z 524.301,A -85,B 0,C 180,E1 14900.282,E2 14900.282} C_VEL
LIN {X 0,Y 386.565,Z 579.919,A -85,B 0,C 180,E1 14898.995,E2 14898.995} C_VEL
LIN {X 0,Y 379.576,Z 636.233,A -85,B 0,C 180,E1 14897.429,E2 14897.429} C_VEL
LIN {X 0,Y 374.411,Z 678.98,A -85,B 0,C 180,E1 14895.921,E2 14895.921} C_VEL
LIN {X 0,Y 371.527,Z 701.631,A -85,B 0,C 180,E1 14894.913,E2 14894.913} C_VEL
LIN {X 0,Y 368.038,Z 722.338,A -85,B 0,C 180,E1 14893.724,E2 14893.724} C_VEL
LIN {X 0,Y 363.901,Z 742.055,A -85,B 0,C 180,E1 14892.314,E2 14892.314} C_VEL
LIN {X 0,Y 359.056,Z 761.63,A -85,B 0,C 180,E1 14890.593,E2 14890.593} C_VEL
LIN {X 0,Y 353.845,Z 779.885,A -85,B 0,C 180,E1 14888.646,E2 14888.646} C_VEL
LIN {X 0,Y 348.221,Z 797.552,A -85,B 0,C 180,E1 14886.367,E2 14886.367} C_VEL
LIN {X 0,Y 342.656,Z 813.579,A -85,B 0,C 180,E1 14883.873,E2 14883.873} C_VEL
LIN {X 0,Y 337.111,Z 828.512,A -85,B 0,C 180,E1 14881.071,E2 14881.071} C_VEL
LIN {X 0,Y 331.922,Z 841.898,A -85,B 0,C 180,E1 14878.03,E2 14878.03} C_VEL
LIN {X 0,Y 327.221,Z 853.771,A -85,B 0,C 180,E1 14874.748,E2 14874.748} C_VEL
LIN {X 0,Y 323.136,Z 864.127,A -85,B 0,C 180,E1 14871.226,E2 14871.226} C_VEL
LIN {X 0,Y 319.793,Z 872.911,A -85,B 0,C 180,E1 14867.467,E2 14867.467} C_VEL
LIN {X 0,Y 317.351,Z 879.758,A -85,B 0,C 180,E1 14863.669,E2 14863.669} C_VEL
LIN {X 0,Y 315.718,Z 884.817,A -85,B 0,C 180,E1 14859.847,E2 14859.847} C_VEL
LIN {X 0,Y 314.775,Z 888.2,A -85,B 0,C 180,E1 14856.017,E2 14856.017} C_VEL
LIN {X 0,Y 314.338,Z 889.944,A -85,B 0,C 180,E1 14852.188,E2 14852.188} C_VEL
LIN {X 0,Y 314.291,Z 890.073,A -85,B 0,C 180,E1 14848.542,E2 14848.542} C_VEL
LIN {X 0,Y 314.639,Z 888.678,A -85,B 0,C 180,E1 14844.712,E2 14844.712} C_VEL
LIN {X 0,Y 315.461,Z 885.688,A -85,B 0,C 180,E1 14840.881,E2 14840.881} C_VEL
LIN {X 0,Y 316.902,Z 881.182,A -85,B 0,C 180,E1 14837.152,E2 14837.152} C_VEL
LIN {X 0,Y 319.088,Z 874.987,A -85,B 0,C 180,E1 14833.432,E2 14833.432} C_VEL
LIN {X 0,Y 322.201,Z 866.746,A -85,B 0,C 180,E1 14829.661,E2 14829.661} C_VEL
LIN {X 0,Y 326.258,Z 856.419,A -85,B 0,C 180,E1 14825.945,E2 14825.945} C_VEL
LIN {X 0,Y 330.771,Z 845.057,A -85,B 0,C 180,E1 14822.646,E2 14822.646} C_VEL
LIN {X 0,Y 335.24,Z 833.575,A -85,B 0,C 180,E1 14819.896,E2 14819.896} C_VEL
LIN {X 0,Y 336.184,Z 829.154,A -85,B 0,C 180,E1 14818.818,E2 14818.818} C_VEL
LIN {X 0,Y 335.663,Z 818.053,A -85,B 0,C 180,E1 14815.965,E2 14815.965} C_VEL
LIN {X 0,Y 336.78,Z 812.978,A -85,B 0,C 180,E1 14814.971,E2 14814.971} C_VEL
LIN {X 0,Y 342.488,Z 797.034,A -85,B 0,C 180,E1 14812.504,E2 14812.504} C_VEL
LIN {X 0,Y 348.159,Z 779.744,A -85,B 0,C 180,E1 14810.282,E2 14810.282} C_VEL
LIN {X 0,Y 353.502,Z 761.486,A -85,B 0,C 180,E1 14808.341,E2 14808.341} C_VEL
LIN {X 0,Y 358.371,Z 742.286,A -85,B 0,C 180,E1 14806.657,E2 14806.657} C_VEL
LIN {X 0,Y 362.464,Z 723.279,A -85,B 0,C 180,E1 14805.296,E2 14805.296} C_VEL
LIN {X 0,Y 365.923,Z 703.4,A -85,B 0,C 180,E1 14804.144,E2 14804.144} C_VEL
LIN {X 0,Y 368.769,Z 681.99,A -85,B 0,C 180,E1 14803.173,E2 14803.173} C_VEL
LIN {X 0,Y 374.11,Z 639.161,A -85,B 0,C 180,E1 14801.628,E2 14801.628} C_VEL
LIN {X 0,Y 380.911,Z 586.596,A -85,B 0,C 180,E1 14800.135,E2 14800.135} C_VEL
LIN {X 0,Y 386.649,Z 533.162,A -85,B 0,C 180,E1 14798.871,E2 14798.871} C_VEL
LIN {X 0,Y 390.901,Z 481.335,A -85,B 0,C 180,E1 14797.84,E2 14797.84} C_VEL
LIN {X 0,Y 394.417,Z 431.388,A -85,B 0,C 180,E1 14796.947,E2 14796.947} C_VEL
LIN {X 0,Y 401.497,Z 400.6,A -85,B 0,C 180,E1 14795.904,E2 14795.904} C_VEL
LIN {X 0,Y 396.31,Z 384.825,A -85,B 0,C 180,E1 14793.195,E2 14793.195} C_VEL
LIN {X 0,Y 390.804,Z 370.04,A -85,B 0,C 180,E1 14790.267,E2 14790.267} C_VEL
LIN {X 0,Y 385.213,Z 356.616,A -85,B 0,C 180,E1 14787.184,E2 14787.184} C_VEL
LIN {X 0,Y 379.626,Z 344.486,A -85,B 0,C 180,E1 14783.889,E2 14783.889} C_VEL
LIN {X 0,Y 374.863,Z 335.107,A -85,B 0,C 180,E1 14780.82,E2 14780.82} C_VEL
LIN {X 0,Y 370.904,Z 327.545,A -85,B 0,C 180,E1 14777.979,E2 14777.979} C_VEL
LIN {X 0,Y 367.713,Z 322.04,A -85,B 0,C 180,E1 14775.455,E2 14775.455} C_VEL
LIN {X 0,Y 365.231,Z 317.579,A -85,B 0,C 180,E1 14773.134,E2 14773.134} C_VEL
LIN {X 0,Y 362.946,Z 313.195,A -85,B 0,C 180,E1 14770.42,E2 14770.42} C_VEL
LIN {X 0,Y 360.105,Z 309.008,A -85,B 0,C 180,E1 14766.617,E2 14766.617} C_VEL
LIN {X 0,Y 359.553,Z 307.196,A -85,B 0,C 180,E1 14765.266,E2 14765.266} C_VEL
LIN {X 0,Y 358.044,Z 305.424,A -85,B 0,C 180,E1 14758.88,E2 14758.88} C_VEL
LIN {X 0,Y 359,Z 306.071,A -85,B 0,C 180,E1 14754.566,E2 14754.566} C_VEL
LIN {X 0,Y 361.012,Z 307.722,A -85,B 0,C 180,E1 14750.997,E2 14750.997} C_VEL
LIN {X 0,Y 363.253,Z 320.836,A -85,B 0,C 180,E1 14746.428,E2 14746.428} C_VEL
LIN {X 0,Y 367.234,Z 334.978,A -85,B 0,C 180,E1 14742.245,E2 14742.245} C_VEL
LIN {X 0,Y 374.146,Z 354.706,A -85,B 0,C 180,E1 14737.366,E2 14737.366} C_VEL
LIN {X 0,Y 378.877,Z 366.831,A -85,B 0,C 180,E1 14734.793,E2 14734.793} C_VEL
LIN {X 0,Y 387.037,Z 388.694,A -85,B 0,C 180,E1 14731.069,E2 14731.069} C_VEL
LIN {X 0,Y 392.039,Z 397.2,A -85,B 0,C 180,E1 14730.094,E2 14730.094} C_VEL
LIN {X 0,Y 364.652,Z 692.358,A -85,B 0,C 180,E1 14722.919,E2 14722.919} C_VEL
LIN {X 0,Y 361.368,Z 717.115,A -85,B 0,C 180,E1 14722.047,E2 14722.047} C_VEL
LIN {X 0,Y 357.136,Z 742.873,A -85,B 0,C 180,E1 14720.853,E2 14720.853} C_VEL
LIN {X 0,Y 352.587,Z 766.526,A -85,B 0,C 180,E1 14719.465,E2 14719.465} C_VEL
LIN {X 0,Y 347.545,Z 789.471,A -85,B 0,C 180,E1 14717.802,E2 14717.802} C_VEL
LIN {X 0,Y 344.555,Z 803.046,A -85,B 0,C 180,E1 14716.752,E2 14716.752} C_VEL
LIN {X 0,Y 340.408,Z 824.125,A -85,B 0,C 180,E1 14715.064,E2 14715.064} C_VEL
LIN {X 0,Y 336.038,Z 843.172,A -85,B 0,C 180,E1 14713.186,E2 14713.186} C_VEL
LIN {X 0,Y 331.289,Z 861.282,A -85,B 0,C 180,E1 14711.014,E2 14711.014} C_VEL
LIN {X 0,Y 326.455,Z 878.195,A -85,B 0,C 180,E1 14708.537,E2 14708.537} C_VEL
LIN {X 0,Y 321.707,Z 893.976,A -85,B 0,C 180,E1 14705.755,E2 14705.755} C_VEL
LIN {X 0,Y 317.312,Z 908.347,A -85,B 0,C 180,E1 14702.716,E2 14702.716} C_VEL
LIN {X 0,Y 313.439,Z 921.294,A -85,B 0,C 180,E1 14699.424,E2 14699.424} C_VEL
LIN {X 0,Y 310.158,Z 933.006,A -85,B 0,C 180,E1 14695.799,E2 14695.799} C_VEL
LIN {X 0,Y 307.705,Z 943.212,A -85,B 0,C 180,E1 14691.944,E2 14691.944} C_VEL
LIN {X 0,Y 306.136,Z 951.866,A -85,B 0,C 180,E1 14687.88,E2 14687.88} C_VEL
LIN {X 0,Y 305.459,Z 958.533,A -85,B 0,C 180,E1 14683.825,E2 14683.825} C_VEL
LIN {X 0,Y 305.478,Z 964.84,A -85,B 0,C 180,E1 14678.849,E2 14678.849} C_VEL
LIN {X 0,Y 305.703,Z 968.418,A -85,B 0,C 180,E1 14675.255,E2 14675.255} C_VEL
LIN {X 0,Y 305.829,Z 970.462,A -85,B 0,C 180,E1 14672.061,E2 14672.061} C_VEL
LIN {X 0,Y 305.756,Z 971.45,A -85,B 0,C 180,E1 14668.688,E2 14668.688} C_VEL
LIN {X 0,Y 305.373,Z 971.154,A -85,B 0,C 180,E1 14664.928,E2 14664.928} C_VEL
LIN {X 0,Y 304.984,Z 969.394,A -85,B 0,C 180,E1 14661.136,E2 14661.136} C_VEL
LIN {X 0,Y 304.909,Z 966.391,A -85,B 0,C 180,E1 14657.308,E2 14657.308} C_VEL
LIN {X 0,Y 305.667,Z 960.934,A -85,B 0,C 180,E1 14652.485,E2 14652.485} C_VEL
LIN {X 0,Y 307.568,Z 954.22,A -85,B 0,C 180,E1 14648.046,E2 14648.046} C_VEL
LIN {X 0,Y 311.587,Z 944.396,A -85,B 0,C 180,E1 14642.891,E2 14642.891} C_VEL
LIN {X 0,Y 317.503,Z 933.001,A -85,B 0,C 180,E1 14638.057,E2 14638.057} C_VEL
LIN {X 0,Y 325.535,Z 919.507,A -85,B 0,C 180,E1 14633.425,E2 14633.425} C_VEL
LIN {X 0,Y 335.726,Z 904.12,A -85,B 0,C 180,E1 14629.063,E2 14629.063} C_VEL
LIN {X 0,Y 347.595,Z 887.511,A -85,B 0,C 180,E1 14625.189,E2 14625.189} C_VEL
LIN {X 0,Y 361.409,Z 869.003,A -85,B 0,C 180,E1 14621.669,E2 14621.669} C_VEL
LIN {X 0,Y 376.495,Z 849.461,A -85,B 0,C 180,E1 14618.666,E2 14618.666} C_VEL
LIN {X 0,Y 383.915,Z 840.004,A -85,B 0,C 180,E1 14617.408,E2 14617.408} C_VEL
LIN {X 0,Y 369.097,Z 854.575,A -85,B 0,C 180,E1 14614.862,E2 14614.862} C_VEL
LIN {X 0,Y 355.676,Z 867.956,A -85,B 0,C 180,E1 14611.905,E2 14611.905} C_VEL
LIN {X 0,Y 343.648,Z 880.049,A -85,B 0,C 180,E1 14608.502,E2 14608.502} C_VEL
LIN {X 0,Y 334.295,Z 889.299,A -85,B 0,C 180,E1 14605.134,E2 14605.134} C_VEL
LIN {X 0,Y 326.776,Z 896.357,A -85,B 0,C 180,E1 14601.731,E2 14601.731} C_VEL
LIN {X 0,Y 320.566,Z 901.556,A -85,B 0,C 180,E1 14598.175,E2 14598.175} C_VEL
LIN {X 0,Y 315.822,Z 904.707,A -85,B 0,C 180,E1 14594.672,E2 14594.672} C_VEL
LIN {X 0,Y 312.335,Z 906.022,A -85,B 0,C 180,E1 14591.261,E2 14591.261} C_VEL
LIN {X 0,Y 309.765,Z 905.647,A -85,B 0,C 180,E1 14587.792,E2 14587.792} C_VEL
LIN {X 0,Y 307.992,Z 903.488,A -85,B 0,C 180,E1 14584.282,E2 14584.282} C_VEL
LIN {X 0,Y 306.93,Z 899.49,A -85,B 0,C 180,E1 14580.747,E2 14580.747} C_VEL
LIN {X 0,Y 306.445,Z 893.956,A -85,B 0,C 180,E1 14577.382,E2 14577.382} C_VEL
LIN {X 0,Y 306.43,Z 886.643,A -85,B 0,C 180,E1 14574.006,E2 14574.006} C_VEL
LIN {X 0,Y 306.843,Z 877.905,A -85,B 0,C 180,E1 14570.812,E2 14570.812} C_VEL
LIN {X 0,Y 307.726,Z 867.204,A -85,B 0,C 180,E1 14567.616,E2 14567.616} C_VEL
LIN {X 0,Y 309.068,Z 855.123,A -85,B 0,C 180,E1 14564.598,E2 14564.598} C_VEL
LIN {X 0,Y 310.917,Z 840.993,A -85,B 0,C 180,E1 14561.629,E2 14561.629} C_VEL
LIN {X 0,Y 313.265,Z 824.574,A -85,B 0,C 180,E1 14558.752,E2 14558.752} C_VEL
LIN {X 0,Y 315.979,Z 806.581,A -85,B 0,C 180,E1 14556.106,E2 14556.106} C_VEL
LIN {X 0,Y 318.981,Z 786.801,A -85,B 0,C 180,E1 14553.679,E2 14553.679} C_VEL
LIN {X 0,Y 322.073,Z 765.694,A -85,B 0,C 180,E1 14551.54,E2 14551.54} C_VEL
LIN {X 0,Y 325.317,Z 742.556,A -85,B 0,C 180,E1 14549.628,E2 14549.628} C_VEL
LIN {X 0,Y 328.168,Z 720.019,A -85,B 0,C 180,E1 14548.138,E2 14548.138} C_VEL
LIN {X 0,Y 330.862,Z 695.808,A -85,B 0,C 180,E1 14546.901,E2 14546.901} C_VEL
LIN {X 0,Y 333.298,Z 668.83,A -85,B 0,C 180,E1 14545.901,E2 14545.901} C_VEL
LIN {X 0,Y 333.951,Z 661.486,A -85,B 0,C 180,E1 14545.64,E2 14545.64} C_VEL
LIN {X 0,Y 335.16,Z 661.308,A -85,B 0,C 180,E1 14545.33,E2 14545.33} C_VEL
LIN {X 0,Y 337.514,Z 658.355,A -85,B 0,C 180,E1 14544.945,E2 14544.945} C_VEL
LIN {X 0,Y 341.352,Z 650.713,A -85,B 0,C 180,E1 14544.537,E2 14544.537} C_VEL
LIN {X 0,Y 345.98,Z 638.87,A -85,B 0,C 180,E1 14544.232,E2 14544.232} C_VEL
LIN {X 0,Y 349.083,Z 635.013,A -85,B 0,C 180,E1 14543.737,E2 14543.737} C_VEL
LIN {X 0,Y 353.01,Z 627.661,A -85,B 0,C 180,E1 14543.298,E2 14543.298} C_VEL
LIN {X 0,Y 357.945,Z 615.208,A -85,B 0,C 180,E1 14542.938,E2 14542.938} C_VEL
LIN {X 0,Y 359.438,Z 611.224,A -85,B 0,C 180,E1 14542.843,E2 14542.843} C_VEL
LIN {X 0,Y 363.279,Z 605.267,A -85,B 0,C 180,E1 14542.335,E2 14542.335} C_VEL
LIN {X 0,Y 367.78,Z 595.544,A -85,B 0,C 180,E1 14541.904,E2 14541.904} C_VEL
LIN {X 0,Y 373.457,Z 579.976,A -85,B 0,C 180,E1 14541.526,E2 14541.526} C_VEL
LIN {X 0,Y 377.822,Z 572.403,A -85,B 0,C 180,E1 14541.009,E2 14541.009} C_VEL
LIN {X 0,Y 382.721,Z 560.896,A -85,B 0,C 180,E1 14540.578,E2 14540.578} C_VEL
LIN {X 0,Y 384.058,Z 557.343,A -85,B 0,C 180,E1 14540.477,E2 14540.477} C_VEL
LIN {X 0,Y 377.756,Z 610.669,A -85,B 0,C 180,E1 14539.108,E2 14539.108} C_VEL
LIN {X 0,Y 371.828,Z 656.088,A -85,B 0,C 180,E1 14537.698,E2 14537.698} C_VEL
LIN {X 0,Y 367.183,Z 693.828,A -85,B 0,C 180,E1 14536.213,E2 14536.213} C_VEL
LIN {X 0,Y 363.852,Z 715.266,A -85,B 0,C 180,E1 14535.092,E2 14535.092} C_VEL
LIN {X 0,Y 359.715,Z 735.954,A -85,B 0,C 180,E1 14533.72,E2 14533.72} C_VEL
LIN {X 0,Y 354.966,Z 755.652,A -85,B 0,C 180,E1 14532.099,E2 14532.099} C_VEL
LIN {X 0,Y 349.776,Z 774.115,A -85,B 0,C 180,E1 14530.245,E2 14530.245} C_VEL
LIN {X 0,Y 344.215,Z 791.654,A -85,B 0,C 180,E1 14528.118,E2 14528.118} C_VEL
LIN {X 0,Y 338.433,Z 808.228,A -85,B 0,C 180,E1 14525.698,E2 14525.698} C_VEL
LIN {X 0,Y 332.607,Z 823.718,A -85,B 0,C 180,E1 14522.965,E2 14522.965} C_VEL
LIN {X 0,Y 327.217,Z 837.285,A -85,B 0,C 180,E1 14520.076,E2 14520.076} C_VEL
LIN {X 0,Y 321.954,Z 850.095,A -85,B 0,C 180,E1 14516.765,E2 14516.765} C_VEL
LIN {X 0,Y 317.521,Z 860.767,A -85,B 0,C 180,E1 14513.377,E2 14513.377} C_VEL
LIN {X 0,Y 313.74,Z 870.01,A -85,B 0,C 180,E1 14509.744,E2 14509.744} C_VEL
LIN {X 0,Y 310.66,Z 877.924,A -85,B 0,C 180,E1 14505.769,E2 14505.769} C_VEL
LIN {X 0,Y 308.519,Z 883.862,A -85,B 0,C 180,E1 14501.782,E2 14501.782} C_VEL
LIN {X 0,Y 307.222,Z 887.941,A -85,B 0,C 180,E1 14497.857,E2 14497.857} C_VEL
LIN {X 0,Y 306.564,Z 890.323,A -85,B 0,C 180,E1 14494.115,E2 14494.115} C_VEL
LIN {X 0,Y 306.339,Z 891.208,A -85,B 0,C 180,E1 14490.187,E2 14490.187} C_VEL
LIN {X 0,Y 306.489,Z 890.546,A -85,B 0,C 180,E1 14486.446,E2 14486.446} C_VEL
LIN {X 0,Y 307.114,Z 888.319,A -85,B 0,C 180,E1 14482.517,E2 14482.517} C_VEL
LIN {X 0,Y 308.332,Z 884.471,A -85,B 0,C 180,E1 14478.591,E2 14478.591} C_VEL
LIN {X 0,Y 310.224,Z 879.232,A -85,B 0,C 180,E1 14474.866,E2 14474.866} C_VEL
LIN {X 0,Y 313.037,Z 871.933,A -85,B 0,C 180,E1 14470.986,E2 14470.986} C_VEL
LIN {X 0,Y 316.625,Z 863.138,A -85,B 0,C 180,E1 14467.339,E2 14467.339} C_VEL
LIN {X 0,Y 321.17,Z 852.205,A -85,B 0,C 180,E1 14463.718,E2 14463.718} C_VEL
LIN {X 0,Y 326.231,Z 839.96,A -85,B 0,C 180,E1 14460.432,E2 14460.432} C_VEL
LIN {X 0,Y 331.829,Z 826.009,A -85,B 0,C 180,E1 14457.359,E2 14457.359} C_VEL
LIN {X 0,Y 336.78,Z 812.978,A -85,B 0,C 180,E1 14454.971,E2 14454.971} C_VEL
LIN {X 0,Y 337.941,Z 807.852,A -85,B 0,C 180,E1 14454,E2 14454} C_VEL
LIN {X 0,Y 338.029,Z 795.096,A -85,B 0,C 180,E1 14451.372,E2 14451.372} C_VEL
LIN {X 0,Y 339.242,Z 789.378,A -85,B 0,C 180,E1 14450.495,E2 14450.495} C_VEL
LIN {X 0,Y 344.718,Z 772.32,A -85,B 0,C 180,E1 14448.476,E2 14448.476} C_VEL
LIN {X 0,Y 349.871,Z 754.202,A -85,B 0,C 180,E1 14446.694,E2 14446.694} C_VEL
LIN {X 0,Y 354.503,Z 735.274,A -85,B 0,C 180,E1 14445.16,E2 14445.16} C_VEL
LIN {X 0,Y 358.506,Z 715.628,A -85,B 0,C 180,E1 14443.865,E2 14443.865} C_VEL
LIN {X 0,Y 361.748,Z 695.38,A -85,B 0,C 180,E1 14442.801,E2 14442.801} C_VEL
LIN {X 0,Y 366.789,Z 656.179,A -85,B 0,C 180,E1 14441.243,E2 14441.243} C_VEL
LIN {X 0,Y 372.959,Z 610.416,A -85,B 0,C 180,E1 14439.817,E2 14439.817} C_VEL
LIN {X 0,Y 379.409,Z 556.738,A -85,B 0,C 180,E1 14438.445,E2 14438.445} C_VEL
LIN {X 0,Y 384.354,Z 505.086,A -85,B 0,C 180,E1 14437.334,E2 14437.334} C_VEL
LIN {X 0,Y 389.545,Z 434.203,A -85,B 0,C 180,E1 14436.046,E2 14436.046} C_VEL
LIN {X 0,Y 396.422,Z 403.987,A -85,B 0,C 180,E1 14435.017,E2 14435.017} C_VEL
LIN {X 0,Y 391.293,Z 388.296,A -85,B 0,C 180,E1 14432.24,E2 14432.24} C_VEL
LIN {X 0,Y 386.296,Z 374.674,A -85,B 0,C 180,E1 14429.459,E2 14429.459} C_VEL
LIN {X 0,Y 380.965,Z 361.708,A -85,B 0,C 180,E1 14426.373,E2 14426.373} C_VEL
LIN {X 0,Y 375.965,Z 350.58,A -85,B 0,C 180,E1 14423.262,E2 14423.262} C_VEL
LIN {X 0,Y 371.595,Z 341.709,A -85,B 0,C 180,E1 14420.311,E2 14420.311} C_VEL
LIN {X 0,Y 367.995,Z 334.569,A -85,B 0,C 180,E1 14417.554,E2 14417.554} C_VEL
LIN {X 0,Y 365.073,Z 329.366,A -85,B 0,C 180,E1 14415.163,E2 14415.163} C_VEL
LIN {X 0,Y 362.77,Z 325.055,A -85,B 0,C 180,E1 14412.901,E2 14412.901} C_VEL
LIN {X 0,Y 360.543,Z 320.629,A -85,B 0,C 180,E1 14410.143,E2 14410.143} C_VEL
LIN {X 0,Y 358.077,Z 316.846,A -85,B 0,C 180,E1 14406.574,E2 14406.574} C_VEL
LIN {X 0,Y 357.526,Z 314.915,A -85,B 0,C 180,E1 14405.135,E2 14405.135} C_VEL
LIN {X 0,Y 356.253,Z 313.222,A -85,B 0,C 180,E1 14398.874,E2 14398.874} C_VEL
LIN {X 0,Y 357.213,Z 313.883,A -85,B 0,C 180,E1 14394.539,E2 14394.539} C_VEL
LIN {X 0,Y 359.144,Z 315.45,A -85,B 0,C 180,E1 14391.273,E2 14391.273} C_VEL
LIN {X 0,Y 361.232,Z 328.608,A -85,B 0,C 180,E1 14386.677,E2 14386.677} C_VEL
LIN {X 0,Y 364.98,Z 342.359,A -85,B 0,C 180,E1 14382.626,E2 14382.626} C_VEL
LIN {X 0,Y 371.783,Z 362.34,A -85,B 0,C 180,E1 14377.673,E2 14377.673} C_VEL
LIN {X 0,Y 375.954,Z 373.486,A -85,B 0,C 180,E1 14375.319,E2 14375.319} C_VEL
LIN {X 0,Y 383.974,Z 396.356,A -85,B 0,C 180,E1 14371.391,E2 14371.391} C_VEL
LIN {X 0,Y 385.536,Z 399.783,A -85,B 0,C 180,E1 14370.861,E2 14370.861} C_VEL
LIN {X 0,Y 385.698,Z 401.009,A -85,B 0,C 180,E1 14370.795,E2 14370.795} C_VEL
LIN {X 0,Y 357.72,Z 692.574,A -85,B 0,C 180,E1 14363.552,E2 14363.552} C_VEL
LIN {X 0,Y 354.365,Z 717.163,A -85,B 0,C 180,E1 14362.666,E2 14362.666} C_VEL
LIN {X 0,Y 350.151,Z 742.267,A -85,B 0,C 180,E1 14361.484,E2 14361.484} C_VEL
LIN {X 0,Y 341.188,Z 789.824,A -85,B 0,C 180,E1 14358.611,E2 14358.611} C_VEL
LIN {X 0,Y 336.274,Z 814.779,A -85,B 0,C 180,E1 14356.76,E2 14356.76} C_VEL
LIN {X 0,Y 331.992,Z 833.623,A -85,B 0,C 180,E1 14355.054,E2 14355.054} C_VEL
LIN {X 0,Y 327.337,Z 851.652,A -85,B 0,C 180,E1 14353.056,E2 14353.056} C_VEL
LIN {X 0,Y 322.418,Z 868.707,A -85,B 0,C 180,E1 14350.754,E2 14350.754} C_VEL
LIN {X 0,Y 317.387,Z 884.838,A -85,B 0,C 180,E1 14348.132,E2 14348.132} C_VEL
LIN {X 0,Y 312.552,Z 900.015,A -85,B 0,C 180,E1 14345.158,E2 14345.158} C_VEL
LIN {X 0,Y 308.132,Z 913.728,A -85,B 0,C 180,E1 14341.933,E2 14341.933} C_VEL
LIN {X 0,Y 304.347,Z 925.934,A -85,B 0,C 180,E1 14338.449,E2 14338.449} C_VEL
LIN {X 0,Y 301.157,Z 937.218,A -85,B 0,C 180,E1 14334.52,E2 14334.52} C_VEL
LIN {X 0,Y 299.026,Z 946.472,A -85,B 0,C 180,E1 14330.555,E2 14330.555} C_VEL
LIN {X 0,Y 297.838,Z 953.879,A -85,B 0,C 180,E1 14326.58,E2 14326.58} C_VEL
LIN {X 0,Y 297.438,Z 959.796,A -85,B 0,C 180,E1 14322.424,E2 14322.424} C_VEL
LIN {X 0,Y 297.642,Z 965.012,A -85,B 0,C 180,E1 14317.528,E2 14317.528} C_VEL
LIN {X 0,Y 297.86,Z 968.051,A -85,B 0,C 180,E1 14314.042,E2 14314.042} C_VEL
LIN {X 0,Y 297.91,Z 969.914,A -85,B 0,C 180,E1 14310.384,E2 14310.384} C_VEL
LIN {X 0,Y 297.666,Z 970.309,A -85,B 0,C 180,E1 14306.726,E2 14306.726} C_VEL
LIN {X 0,Y 297.231,Z 969.515,A -85,B 0,C 180,E1 14303.238,E2 14303.238} C_VEL
LIN {X 0,Y 296.919,Z 967.523,A -85,B 0,C 180,E1 14299.522,E2 14299.522} C_VEL
LIN {X 0,Y 297.166,Z 963.42,A -85,B 0,C 180,E1 14294.784,E2 14294.784} C_VEL
LIN {X 0,Y 298.467,Z 957.805,A -85,B 0,C 180,E1 14290.223,E2 14290.223} C_VEL
LIN {X 0,Y 301.528,Z 949.695,A -85,B 0,C 180,E1 14285.093,E2 14285.093} C_VEL
LIN {X 0,Y 306.392,Z 940.012,A -85,B 0,C 180,E1 14280.236,E2 14280.236} C_VEL
LIN {X 0,Y 313.805,Z 927.706,A -85,B 0,C 180,E1 14275.225,E2 14275.225} C_VEL
LIN {X 0,Y 323.243,Z 913.972,A -85,B 0,C 180,E1 14270.644,E2 14270.644} C_VEL
LIN {X 0,Y 334.892,Z 898.353,A -85,B 0,C 180,E1 14266.394,E2 14266.394} C_VEL
LIN {X 0,Y 348.712,Z 880.922,A -85,B 0,C 180,E1 14262.53,E2 14262.53} C_VEL
LIN {X 0,Y 364.003,Z 862.509,A -85,B 0,C 180,E1 14259.228,E2 14259.228} C_VEL
LIN {X 0,Y 374.502,Z 850.087,A -85,B 0,C 180,E1 14257.354,E2 14257.354} C_VEL
LIN {X 0,Y 359.179,Z 863.893,A -85,B 0,C 180,E1 14254.604,E2 14254.604} C_VEL
LIN {X 0,Y 345.39,Z 876.409,A -85,B 0,C 180,E1 14251.406,E2 14251.406} C_VEL
LIN {X 0,Y 334.044,Z 886.682,A -85,B 0,C 180,E1 14248.031,E2 14248.031} C_VEL
LIN {X 0,Y 324.816,Z 894.747,A -85,B 0,C 180,E1 14244.556,E2 14244.556} C_VEL
LIN {X 0,Y 317.429,Z 900.711,A -85,B 0,C 180,E1 14241.045,E2 14241.045} C_VEL
LIN {X 0,Y 311.375,Z 904.852,A -85,B 0,C 180,E1 14237.376,E2 14237.376} C_VEL
LIN {X 0,Y 306.614,Z 907.076,A -85,B 0,C 180,E1 14233.58,E2 14233.58} C_VEL
LIN {X 0,Y 303.223,Z 907.337,A -85,B 0,C 180,E1 14229.873,E2 14229.873} C_VEL
LIN {X 0,Y 300.934,Z 905.842,A -85,B 0,C 180,E1 14226.295,E2 14226.295} C_VEL
LIN {X 0,Y 299.448,Z 902.582,A -85,B 0,C 180,E1 14222.679,E2 14222.679} C_VEL
LIN {X 0,Y 298.646,Z 897.473,A -85,B 0,C 180,E1 14219.041,E2 14219.041} C_VEL
LIN {X 0,Y 298.396,Z 890.829,A -85,B 0,C 180,E1 14215.58,E2 14215.58} C_VEL
LIN {X 0,Y 298.637,Z 882.294,A -85,B 0,C 180,E1 14212.11,E2 14212.11} C_VEL
LIN {X 0,Y 299.334,Z 872.343,A -85,B 0,C 180,E1 14208.829,E2 14208.829} C_VEL
LIN {X 0,Y 300.57,Z 860.253,A -85,B 0,C 180,E1 14205.552,E2 14205.552} C_VEL
LIN {X 0,Y 302.28,Z 846.733,A -85,B 0,C 180,E1 14202.481,E2 14202.481} C_VEL
LIN {X 0,Y 304.571,Z 830.787,A -85,B 0,C 180,E1 14199.435,E2 14199.435} C_VEL
LIN {X 0,Y 307.18,Z 813.682,A -85,B 0,C 180,E1 14196.703,E2 14196.703} C_VEL
LIN {X 0,Y 310.097,Z 794.889,A -85,B 0,C 180,E1 14194.195,E2 14194.195} C_VEL
LIN {X 0,Y 313.218,Z 774.353,A -85,B 0,C 180,E1 14191.909,E2 14191.909} C_VEL
LIN {X 0,Y 316.543,Z 751.825,A -85,B 0,C 180,E1 14189.851,E2 14189.851} C_VEL
LIN {X 0,Y 319.689,Z 728.685,A -85,B 0,C 180,E1 14188.143,E2 14188.143} C_VEL
LIN {X 0,Y 322.597,Z 704.405,A -85,B 0,C 180,E1 14186.748,E2 14186.748} C_VEL
LIN {X 0,Y 324.402,Z 688.186,A -85,B 0,C 180,E1 14185.984,E2 14185.984} C_VEL
LIN {X 0,Y 325.636,Z 688.059,A -85,B 0,C 180,E1 14185.652,E2 14185.652} C_VEL
LIN {X 0,Y 327.891,Z 685.502,A -85,B 0,C 180,E1 14185.259,E2 14185.259} C_VEL
LIN {X 0,Y 331.75,Z 678.48,A -85,B 0,C 180,E1 14184.827,E2 14184.827} C_VEL
LIN {X 0,Y 336.333,Z 667.667,A -85,B 0,C 180,E1 14184.517,E2 14184.517} C_VEL
LIN {X 0,Y 339.475,Z 663.92,A -85,B 0,C 180,E1 14184.012,E2 14184.012} C_VEL
LIN {X 0,Y 343.394,Z 656.895,A -85,B 0,C 180,E1 14183.571,E2 14183.571} C_VEL
LIN {X 0,Y 348.297,Z 645.248,A -85,B 0,C 180,E1 14183.228,E2 14183.228} C_VEL
LIN {X 0,Y 349.24,Z 643.212,A -85,B 0,C 180,E1 14183.144,E2 14183.144} C_VEL
LIN {X 0,Y 353.089,Z 637.648,A -85,B 0,C 180,E1 14182.621,E2 14182.621} C_VEL
LIN {X 0,Y 357.645,Z 628.586,A -85,B 0,C 180,E1 14182.182,E2 14182.182} C_VEL
LIN {X 0,Y 363.002,Z 615.103,A -85,B 0,C 180,E1 14181.826,E2 14181.826} C_VEL
LIN {X 0,Y 367.492,Z 607.691,A -85,B 0,C 180,E1 14181.297,E2 14181.297} C_VEL
LIN {X 0,Y 372.393,Z 596.823,A -85,B 0,C 180,E1 14180.877,E2 14180.877} C_VEL
LIN {X 0,Y 375.613,Z 588.328,A -85,B 0,C 180,E1 14180.668,E2 14180.668} C_VEL
LIN {X 0,Y 368.648,Z 640.972,A -85,B 0,C 180,E1 14179.163,E2 14179.163} C_VEL
LIN {X 0,Y 363.114,Z 683.795,A -85,B 0,C 180,E1 14177.591,E2 14177.591} C_VEL
LIN {X 0,Y 360.052,Z 705.878,A -85,B 0,C 180,E1 14176.569,E2 14176.569} C_VEL
LIN {X 0,Y 356.301,Z 726.402,A -85,B 0,C 180,E1 14175.349,E2 14175.349} C_VEL
LIN {X 0,Y 351.864,Z 746.01,A -85,B 0,C 180,E1 14173.898,E2 14173.898} C_VEL
LIN {X 0,Y 346.634,Z 765.549,A -85,B 0,C 180,E1 14172.119,E2 14172.119} C_VEL
LIN {X 0,Y 340.825,Z 784.337,A -85,B 0,C 180,E1 14170.03,E2 14170.03} C_VEL
LIN {X 0,Y 334.834,Z 801.656,A -85,B 0,C 180,E1 14167.688,E2 14167.688} C_VEL
LIN {X 0,Y 328.814,Z 817.581,A -85,B 0,C 180,E1 14165.081,E2 14165.081} C_VEL
LIN {X 0,Y 322.895,Z 832.224,A -85,B 0,C 180,E1 14162.183,E2 14162.183} C_VEL
LIN {X 0,Y 317.342,Z 845.359,A -85,B 0,C 180,E1 14159.028,E2 14159.028} C_VEL
LIN {X 0,Y 312.298,Z 857,A -85,B 0,C 180,E1 14155.609,E2 14155.609} C_VEL
LIN {X 0,Y 307.902,Z 867.134,A -85,B 0,C 180,E1 14151.929,E2 14151.929} C_VEL
LIN {X 0,Y 304.295,Z 875.703,A -85,B 0,C 180,E1 14147.992,E2 14147.992} C_VEL
LIN {X 0,Y 301.659,Z 882.344,A -85,B 0,C 180,E1 14144.003,E2 14144.003} C_VEL
LIN {X 0,Y 299.834,Z 887.403,A -85,B 0,C 180,E1 14139.792,E2 14139.792} C_VEL
LIN {X 0,Y 298.86,Z 890.521,A -85,B 0,C 180,E1 14135.761,E2 14135.761} C_VEL
LIN {X 0,Y 298.446,Z 892.023,A -85,B 0,C 180,E1 14131.92,E2 14131.92} C_VEL
LIN {X 0,Y 298.441,Z 892.036,A -85,B 0,C 180,E1 14128.08,E2 14128.08} C_VEL
LIN {X 0,Y 298.847,Z 890.585,A -85,B 0,C 180,E1 14124.239,E2 14124.239} C_VEL
LIN {X 0,Y 299.808,Z 887.52,A -85,B 0,C 180,E1 14120.207,E2 14120.207} C_VEL
LIN {X 0,Y 301.515,Z 882.791,A -85,B 0,C 180,E1 14116.186,E2 14116.186} C_VEL
LIN {X 0,Y 303.952,Z 876.657,A -85,B 0,C 180,E1 14112.384,E2 14112.384} C_VEL
LIN {X 0,Y 307.265,Z 868.804,A -85,B 0,C 180,E1 14108.625,E2 14108.625} C_VEL
LIN {X 0,Y 311.499,Z 859.044,A -85,B 0,C 180,E1 14104.931,E2 14104.931} C_VEL
LIN {X 0,Y 316.674,Z 847.142,A -85,B 0,C 180,E1 14101.319,E2 14101.319} C_VEL
LIN {X 0,Y 322.136,Z 834.333,A -85,B 0,C 180,E1 14098.152,E2 14098.152} C_VEL
LIN {X 0,Y 327.967,Z 820.047,A -85,B 0,C 180,E1 14095.242,E2 14095.242} C_VEL
LIN {X 0,Y 334.223,Z 803.699,A -85,B 0,C 180,E1 14092.497,E2 14092.497} C_VEL
LIN {X 0,Y 339.242,Z 789.378,A -85,B 0,C 180,E1 14090.495,E2 14090.495} C_VEL
LIN {X 0,Y 340.475,Z 783.625,A -85,B 0,C 180,E1 14089.641,E2 14089.641} C_VEL
LIN {X 0,Y 340.769,Z 769.373,A -85,B 0,C 180,E1 14087.274,E2 14087.274} C_VEL
LIN {X 0,Y 341.959,Z 763.048,A -85,B 0,C 180,E1 14086.517,E2 14086.517} C_VEL
LIN {X 0,Y 346.995,Z 744.339,A -85,B 0,C 180,E1 14084.857,E2 14084.857} C_VEL
LIN {X 0,Y 351.352,Z 725.232,A -85,B 0,C 180,E1 14083.474,E2 14083.474} C_VEL
LIN {X 0,Y 355.11,Z 704.688,A -85,B 0,C 180,E1 14082.276,E2 14082.276} C_VEL
LIN {X 0,Y 358.615,Z 679.329,A -85,B 0,C 180,E1 14081.141,E2 14081.141} C_VEL
LIN {X 0,Y 364.283,Z 637.626,A -85,B 0,C 180,E1 14079.638,E2 14079.638} C_VEL
LIN {X 0,Y 371.135,Z 586.782,A -85,B 0,C 180,E1 14078.201,E2 14078.201} C_VEL
LIN {X 0,Y 377.109,Z 533.395,A -85,B 0,C 180,E1 14076.942,E2 14076.942} C_VEL
LIN {X 0,Y 381.368,Z 483.071,A -85,B 0,C 180,E1 14075.947,E2 14075.947} C_VEL
LIN {X 0,Y 384.825,Z 436.662,A -85,B 0,C 180,E1 14075.113,E2 14075.113} C_VEL
LIN {X 0,Y 391.487,Z 407.522,A -85,B 0,C 180,E1 14074.128,E2 14074.128} C_VEL
LIN {X 0,Y 386.519,Z 392.199,A -85,B 0,C 180,E1 14071.33,E2 14071.33} C_VEL
LIN {X 0,Y 381.381,Z 378.048,A -85,B 0,C 180,E1 14068.33,E2 14068.33} C_VEL
LIN {X 0,Y 376.23,Z 365.361,A -85,B 0,C 180,E1 14065.165,E2 14065.165} C_VEL
LIN {X 0,Y 371.348,Z 354.346,A -85,B 0,C 180,E1 14061.896,E2 14061.896} C_VEL
LIN {X 0,Y 367.077,Z 345.55,A -85,B 0,C 180,E1 14058.749,E2 14058.749} C_VEL
LIN {X 0,Y 364.606,Z 340.77,A -85,B 0,C 180,E1 14056.735,E2 14056.735} C_VEL
LIN {X 0,Y 362.517,Z 336.712,A -85,B 0,C 180,E1 14054.863,E2 14054.863} C_VEL
LIN {X 0,Y 360.35,Z 332.462,A -85,B 0,C 180,E1 14052.581,E2 14052.581} C_VEL
LIN {X 0,Y 357.865,Z 327.689,A -85,B 0,C 180,E1 14049.489,E2 14049.489} C_VEL
LIN {X 0,Y 355.935,Z 324.353,A -85,B 0,C 180,E1 14046.29,E2 14046.29} C_VEL
LIN {X 0,Y 355.5,Z 322.634,A -85,B 0,C 180,E1 14045.002,E2 14045.002} C_VEL
LIN {X 0,Y 354.47,Z 320.986,A -85,B 0,C 180,E1 14038.545,E2 14038.545} C_VEL
LIN {X 0,Y 355.671,Z 321.876,A -85,B 0,C 180,E1 14034.029,E2 14034.029} C_VEL
LIN {X 0,Y 357.257,Z 323.157,A -85,B 0,C 180,E1 14031.551,E2 14031.551} C_VEL
LIN {X 0,Y 359.098,Z 335.798,A -85,B 0,C 180,E1 14027.129,E2 14027.129} C_VEL
LIN {X 0,Y 362.564,Z 349.288,A -85,B 0,C 180,E1 14023.13,E2 14023.13} C_VEL
LIN {X 0,Y 369.014,Z 369.011,A -85,B 0,C 180,E1 14018.209,E2 14018.209} C_VEL
LIN {X 0,Y 372.901,Z 379.636,A -85,B 0,C 180,E1 14015.948,E2 14015.948} C_VEL
LIN {X 0,Y 380.695,Z 402.746,A -85,B 0,C 180,E1 14011.935,E2 14011.935} C_VEL
LIN {X 0,Y 381.092,Z 404.189,A -85,B 0,C 180,E1 14011.735,E2 14011.735} C_VEL
LIN {X 0,Y 363.956,Z 554.058,A -85,B 0,C 180,E1 14007.843,E2 14007.843} C_VEL
LIN {X 0,Y 358.565,Z 611.238,A -85,B 0,C 180,E1 14006.408,E2 14006.408} C_VEL
LIN {X 0,Y 355.678,Z 653.164,A -85,B 0,C 180,E1 14005.509,E2 14005.509} C_VEL
LIN {X 0,Y 352.116,Z 687.641,A -85,B 0,C 180,E1 14004.527,E2 14004.527} C_VEL
LIN {X 0,Y 347.408,Z 721.446,A -85,B 0,C 180,E1 14003.297,E2 14003.297} C_VEL
LIN {X 0,Y 342.681,Z 750.705,A -85,B 0,C 180,E1 14001.917,E2 14001.917} C_VEL
LIN {X 0,Y 337.211,Z 780.861,A -85,B 0,C 180,E1 14000.172,E2 14000.172} C_VEL
LIN {X 0,Y 331.507,Z 809.252,A -85,B 0,C 180,E1 13998.159,E2 13998.159} C_VEL
LIN {X 0,Y 327.245,Z 827.893,A -85,B 0,C 180,E1 13996.525,E2 13996.525} C_VEL
LIN {X 0,Y 322.518,Z 845.852,A -85,B 0,C 180,E1 13994.604,E2 13994.604} C_VEL
LIN {X 0,Y 317.602,Z 862.404,A -85,B 0,C 180,E1 13992.477,E2 13992.477} C_VEL
LIN {X 0,Y 312.385,Z 878.87,A -85,B 0,C 180,E1 13989.924,E2 13989.924} C_VEL
LIN {X 0,Y 307.204,Z 894.344,A -85,B 0,C 180,E1 13987.023,E2 13987.023} C_VEL
LIN {X 0,Y 302.284,Z 908.668,A -85,B 0,C 180,E1 13983.759,E2 13983.759} C_VEL
LIN {X 0,Y 297.991,Z 921.531,A -85,B 0,C 180,E1 13980.219,E2 13980.219} C_VEL
LIN {X 0,Y 294.466,Z 932.94,A -85,B 0,C 180,E1 13976.412,E2 13976.412} C_VEL
LIN {X 0,Y 291.816,Z 942.875,A -85,B 0,C 180,E1 13972.31,E2 13972.31} C_VEL
LIN {X 0,Y 290.161,Z 951.193,A -85,B 0,C 180,E1 13967.993,E2 13967.993} C_VEL
LIN {X 0,Y 289.494,Z 957.489,A -85,B 0,C 180,E1 13963.787,E2 13963.787} C_VEL
LIN {X 0,Y 289.553,Z 962.147,A -85,B 0,C 180,E1 13959.541,E2 13959.541} C_VEL
LIN {X 0,Y 289.9,Z 965.745,A -85,B 0,C 180,E1 13955.343,E2 13955.343} C_VEL
LIN {X 0,Y 290.044,Z 968.016,A -85,B 0,C 180,E1 13951.778,E2 13951.778} C_VEL
LIN {X 0,Y 289.94,Z 968.994,A -85,B 0,C 180,E1 13948.617,E2 13948.617} C_VEL
LIN {X 0,Y 289.558,Z 968.983,A -85,B 0,C 180,E1 13945.246,E2 13945.246} C_VEL
LIN {X 0,Y 289.099,Z 967.8,A -85,B 0,C 180,E1 13941.447,E2 13941.447} C_VEL
LIN {X 0,Y 288.987,Z 964.607,A -85,B 0,C 180,E1 13936.596,E2 13936.596} C_VEL
LIN {X 0,Y 289.757,Z 960.148,A -85,B 0,C 180,E1 13932.114,E2 13932.114} C_VEL
LIN {X 0,Y 292.21,Z 953.138,A -85,B 0,C 180,E1 13926.827,E2 13926.827} C_VEL
LIN {X 0,Y 296.428,Z 944.613,A -85,B 0,C 180,E1 13921.82,E2 13921.82} C_VEL
LIN {X 0,Y 303.398,Z 933.28,A -85,B 0,C 180,E1 13916.491,E2 13916.491} C_VEL
LIN {X 0,Y 312.593,Z 920.465,A -85,B 0,C 180,E1 13911.599,E2 13911.599} C_VEL
LIN {X 0,Y 324.233,Z 905.701,A -85,B 0,C 180,E1 13907.036,E2 13907.036} C_VEL
LIN {X 0,Y 338.331,Z 889.038,A -85,B 0,C 180,E1 13902.867,E2 13902.867} C_VEL
LIN {X 0,Y 354.739,Z 870.663,A -85,B 0,C 180,E1 13899.183,E2 13899.183} C_VEL
LIN {X 0,Y 365.018,Z 859.44,A -85,B 0,C 180,E1 13897.301,E2 13897.301} C_VEL
LIN {X 0,Y 349.209,Z 872.446,A -85,B 0,C 180,E1 13894.338,E2 13894.338} C_VEL
LIN {X 0,Y 335.594,Z 883.653,A -85,B 0,C 180,E1 13891.028,E2 13891.028} C_VEL
LIN {X 0,Y 324.384,Z 892.704,A -85,B 0,C 180,E1 13887.54,E2 13887.54} C_VEL
LIN {X 0,Y 315.292,Z 899.629,A -85,B 0,C 180,E1 13883.949,E2 13883.949} C_VEL
LIN {X 0,Y 308.049,Z 904.537,A -85,B 0,C 180,E1 13880.323,E2 13880.323} C_VEL
LIN {X 0,Y 302.172,Z 907.645,A -85,B 0,C 180,E1 13876.533,E2 13876.533} C_VEL
LIN {X 0,Y 297.811,Z 908.844,A -85,B 0,C 180,E1 13872.803,E2 13872.803} C_VEL
LIN {X 0,Y 294.664,Z 908.287,A -85,B 0,C 180,E1 13869.083,E2 13869.083} C_VEL
LIN {X 0,Y 292.468,Z 905.923,A -85,B 0,C 180,E1 13865.296,E2 13865.296} C_VEL
LIN {X 0,Y 291.159,Z 901.801,A -85,B 0,C 180,E1 13861.574,E2 13861.574} C_VEL
LIN {X 0,Y 290.513,Z 895.812,A -85,B 0,C 180,E1 13857.83,E2 13857.83} C_VEL
LIN {X 0,Y 290.44,Z 888.231,A -85,B 0,C 180,E1 13854.231,E2 13854.231} C_VEL
LIN {X 0,Y 290.873,Z 878.851,A -85,B 0,C 180,E1 13850.702,E2 13850.702} C_VEL
LIN {X 0,Y 291.811,Z 867.931,A -85,B 0,C 180,E1 13847.332,E2 13847.332} C_VEL
LIN {X 0,Y 293.234,Z 855.611,A -85,B 0,C 180,E1 13844.17,E2 13844.17} C_VEL
LIN {X 0,Y 295.081,Z 841.982,A -85,B 0,C 180,E1 13841.221,E2 13841.221} C_VEL
LIN {X 0,Y 297.464,Z 826.09,A -85,B 0,C 180,E1 13838.3,E2 13838.3} C_VEL
LIN {X 0,Y 300.213,Z 808.748,A -85,B 0,C 180,E1 13835.607,E2 13835.607} C_VEL
LIN {X 0,Y 303.242,Z 789.904,A -85,B 0,C 180,E1 13833.145,E2 13833.145} C_VEL
LIN {X 0,Y 306.442,Z 769.276,A -85,B 0,C 180,E1 13830.91,E2 13830.91} C_VEL
LIN {X 0,Y 309.807,Z 746.584,A -85,B 0,C 180,E1 13828.909,E2 13828.909} C_VEL
LIN {X 0,Y 313.021,Z 722.706,A -85,B 0,C 180,E1 13827.218,E2 13827.218} C_VEL
LIN {X 0,Y 314.397,Z 711.79,A -85,B 0,C 180,E1 13826.565,E2 13826.565} C_VEL
LIN {X 0,Y 315.558,Z 711.842,A -85,B 0,C 180,E1 13826.213,E2 13826.213} C_VEL
LIN {X 0,Y 317.977,Z 709.611,A -85,B 0,C 180,E1 13825.745,E2 13825.745} C_VEL
LIN {X 0,Y 321.775,Z 703.882,A -85,B 0,C 180,E1 13825.262,E2 13825.262} C_VEL
LIN {X 0,Y 326.016,Z 695.125,A -85,B 0,C 180,E1 13824.909,E2 13824.909} C_VEL
LIN {X 0,Y 329.867,Z 690.849,A -85,B 0,C 180,E1 13824.276,E2 13824.276} C_VEL
LIN {X 0,Y 333.975,Z 683.923,A -85,B 0,C 180,E1 13823.804,E2 13823.804} C_VEL
LIN {X 0,Y 338.441,Z 674.02,A -85,B 0,C 180,E1 13823.486,E2 13823.486} C_VEL
LIN {X 0,Y 339.39,Z 672.118,A -85,B 0,C 180,E1 13823.4,E2 13823.4} C_VEL
LIN {X 0,Y 343.392,Z 666.592,A -85,B 0,C 180,E1 13822.855,E2 13822.855} C_VEL
LIN {X 0,Y 348.05,Z 657.692,A -85,B 0,C 180,E1 13822.411,E2 13822.411} C_VEL
LIN {X 0,Y 352.501,Z 647.411,A -85,B 0,C 180,E1 13822.112,E2 13822.112} C_VEL
LIN {X 0,Y 357.058,Z 640.454,A -85,B 0,C 180,E1 13821.561,E2 13821.561} C_VEL
LIN {X 0,Y 362.014,Z 630.337,A -85,B 0,C 180,E1 13821.13,E2 13821.13} C_VEL
